LIN {X 0,Y 468.633,Z 235.957,A -85,B 0,C 180,E1 -7687.941,E2 -7687.941} C_VEL
LIN {X 0,Y 467.587,Z 230.243,A -85,B 0,C 180,E1 -7690.829,E2 -7690.829} C_VEL
LIN {X 0,Y 467.551,Z 230.247,A -85,B 0,C 180,E1 -7693.819,E2 -7693.819} C_VEL
LIN {X 0,Y 467.553,Z 230.248,A -85,B 0,C 180,E1 -7696.254,E2 -7696.254} C_VEL
LIN {X 0,Y 467.577,Z 230.245,A -85,B 0,C 180,E1 -7698.722,E2 -7698.722} C_VEL
LIN {X 0,Y 467.564,Z 230.246,A -85,B 0,C 180,E1 -7701.954,E2 -7701.954} C_VEL
LIN {X 0,Y 467.566,Z 230.245,A -85,B 0,C 180,E1 -7705.166,E2 -7705.166} C_VEL
LIN {X 0,Y 467.581,Z 230.243,A -85,B 0,C 180,E1 -7708.259,E2 -7708.259} C_VEL
LIN {X 0,Y 467.575,Z 230.245,A -85,B 0,C 180,E1 -7711.249,E2 -7711.249} C_VEL
LIN {X 0,Y 467.61,Z 230.239,A -85,B 0,C 180,E1 -7713.198,E2 -7713.198} C_VEL
LIN {X 0,Y 467.587,Z 230.242,A -85,B 0,C 180,E1 -7716.467,E2 -7716.467} C_VEL
LIN {X 0,Y 467.621,Z 230.237,A -85,B 0,C 180,E1 -7719.776,E2 -7719.776} C_VEL
LIN {X 0,Y 467.605,Z 230.241,A -85,B 0,C 180,E1 -7722.505,E2 -7722.505} C_VEL
LIN {X 0,Y 467.603,Z 230.24,A -85,B 0,C 180,E1 -7725.195,E2 -7725.195} C_VEL
LIN {X 0,Y 467.679,Z 230.23,A -85,B 0,C 180,E1 -7727.854,E2 -7727.854} C_VEL
LIN {X 0,Y 467.677,Z 230.231,A -85,B 0,C 180,E1 -7731.356,E2 -7731.356} C_VEL
LIN {X 0,Y 467.739,Z 230.225,A -85,B 0,C 180,E1 -7733.961,E2 -7733.961} C_VEL
LIN {X 0,Y 467.855,Z 230.21,A -85,B 0,C 180,E1 -7737.416,E2 -7737.416} C_VEL
LIN {X 0,Y 467.876,Z 230.206,A -85,B 0,C 180,E1 -7739.999,E2 -7739.999} C_VEL
LIN {X 0,Y 467.855,Z 230.208,A -85,B 0,C 180,E1 -7742.582,E2 -7742.582} C_VEL
LIN {X 0,Y 467.737,Z 230.224,A -85,B 0,C 180,E1 -7746.036,E2 -7746.036} C_VEL
LIN {X 0,Y 467.676,Z 230.232,A -85,B 0,C 180,E1 -7748.641,E2 -7748.641} C_VEL
LIN {X 0,Y 467.682,Z 230.231,A -85,B 0,C 180,E1 -7752.378,E2 -7752.378} C_VEL
LIN {X 0,Y 467.639,Z 230.239,A -85,B 0,C 180,E1 -7755.884,E2 -7755.884} C_VEL
LIN {X 0,Y 467.425,Z 230.265,A -85,B 0,C 180,E1 -7758.698,E2 -7758.698} C_VEL
LIN {X 0,Y 467.242,Z 230.477,A -85,B 0,C 180,E1 -7760.238,E2 -7760.238} C_VEL
LIN {X 0,Y 467.196,Z 233.681,A -85,B 0,C 180,E1 -7763.422,E2 -7763.422} C_VEL
LIN {X 0,Y 467.086,Z 236.163,A -85,B 0,C 180,E1 -7765.869,E2 -7765.869} C_VEL
LIN {X 0,Y 467.03,Z 239.651,A -85,B 0,C 180,E1 -7769.216,E2 -7769.216} C_VEL
LIN {X 0,Y 466.954,Z 242.322,A -85,B 0,C 180,E1 -7771.786,E2 -7771.786} C_VEL
LIN {X 0,Y 466.836,Z 245.609,A -85,B 0,C 180,E1 -7774.893,E2 -7774.893} C_VEL
LIN {X 0,Y 466.815,Z 248.588,A -85,B 0,C 180,E1 -7777.682,E2 -7777.682} C_VEL
LIN {X 0,Y 470.307,Z 263.21,A -85,B 0,C 180,E1 -7778.274,E2 -7778.274} C_VEL
LIN {X 0,Y 470.1,Z 275.079,A -85,B 0,C 180,E1 -7778.817,E2 -7778.817} C_VEL
LIN {X 0,Y 469.595,Z 287.366,A -85,B 0,C 180,E1 -7779.565,E2 -7779.565} C_VEL
LIN {X 0,Y 469.105,Z 298.069,A -85,B 0,C 180,E1 -7780.398,E2 -7780.398} C_VEL
LIN {X 0,Y 468.677,Z 308.639,A -85,B 0,C 180,E1 -7781.431,E2 -7781.431} C_VEL
LIN {X 0,Y 468.115,Z 318.546,A -85,B 0,C 180,E1 -7782.639,E2 -7782.639} C_VEL
LIN {X 0,Y 467.709,Z 326.533,A -85,B 0,C 180,E1 -7783.842,E2 -7783.842} C_VEL
LIN {X 0,Y 467.423,Z 332.988,A -85,B 0,C 180,E1 -7785.036,E2 -7785.036} C_VEL
LIN {X 0,Y 467.098,Z 339.332,A -85,B 0,C 180,E1 -7786.517,E2 -7786.517} C_VEL
LIN {X 0,Y 466.899,Z 344.209,A -85,B 0,C 180,E1 -7788.019,E2 -7788.019} C_VEL
LIN {X 0,Y 466.732,Z 347.944,A -85,B 0,C 180,E1 -7789.649,E2 -7789.649} C_VEL
LIN {X 0,Y 466.651,Z 349.597,A -85,B 0,C 180,E1 -7790.763,E2 -7790.763} C_VEL
LIN {X 0,Y 466.585,Z 350.586,A -85,B 0,C 180,E1 -7791.863,E2 -7791.863} C_VEL
LIN {X 0,Y 466.563,Z 350.949,A -85,B 0,C 180,E1 -7792.97,E2 -7792.97} C_VEL
LIN {X 0,Y 466.58,Z 350.427,A -85,B 0,C 180,E1 -7794.425,E2 -7794.425} C_VEL
LIN {X 0,Y 466.705,Z 348.328,A -85,B 0,C 180,E1 -7796.141,E2 -7796.141} C_VEL
LIN {X 0,Y 466.812,Z 345.614,A -85,B 0,C 180,E1 -7797.465,E2 -7797.465} C_VEL
LIN {X 0,Y 467.018,Z 340.95,A -85,B 0,C 180,E1 -7799.064,E2 -7799.064} C_VEL
LIN {X 0,Y 467.287,Z 335.172,A -85,B 0,C 180,E1 -7800.522,E2 -7800.522} C_VEL
LIN {X 0,Y 467.632,Z 327.673,A -85,B 0,C 180,E1 -7801.989,E2 -7801.989} C_VEL
LIN {X 0,Y 468.024,Z 319.77,A -85,B 0,C 180,E1 -7803.226,E2 -7803.226} C_VEL
LIN {X 0,Y 468.415,Z 311.541,A -85,B 0,C 180,E1 -7804.279,E2 -7804.279} C_VEL
LIN {X 0,Y 468.893,Z 301.772,A -85,B 0,C 180,E1 -7805.3,E2 -7805.3} C_VEL
LIN {X 0,Y 469.394,Z 290.021,A -85,B 0,C 180,E1 -7806.286,E2 -7806.286} C_VEL
LIN {X 0,Y 469.167,Z 284.982,A -85,B 0,C 180,E1 -7806.654,E2 -7806.654} C_VEL
LIN {X 0,Y 467.195,Z 276.584,A -85,B 0,C 180,E1 -7807.24,E2 -7807.24} C_VEL
LIN {X 0,Y 465.004,Z 269.763,A -85,B 0,C 180,E1 -7807.668,E2 -7807.668} C_VEL
LIN {X 0,Y 463.062,Z 262.658,A -85,B 0,C 180,E1 -7808.038,E2 -7808.038} C_VEL
LIN {X 0,Y 460.055,Z 249.852,A -85,B 0,C 180,E1 -7808.552,E2 -7808.552} C_VEL
LIN {X 0,Y 459.77,Z 248.251,A -85,B 0,C 180,E1 -7808.628,E2 -7808.628} C_VEL
LIN {X 0,Y 459.812,Z 245.224,A -85,B 0,C 180,E1 -7811.37,E2 -7811.37} C_VEL
LIN {X 0,Y 459.898,Z 242.015,A -85,B 0,C 180,E1 -7814.303,E2 -7814.303} C_VEL
LIN {X 0,Y 459.964,Z 238.118,A -85,B 0,C 180,E1 -7817.918,E2 -7817.918} C_VEL
LIN {X 0,Y 460.035,Z 234.635,A -85,B 0,C 180,E1 -7821.213,E2 -7821.213} C_VEL
LIN {X 0,Y 460.077,Z 231.831,A -85,B 0,C 180,E1 -7823.863,E2 -7823.863} C_VEL
LIN {X 0,Y 460.173,Z 231.168,A -85,B 0,C 180,E1 -7824.743,E2 -7824.743} C_VEL
LIN {X 0,Y 460.662,Z 231.104,A -85,B 0,C 180,E1 -7828.252,E2 -7828.252} C_VEL
LIN {X 0,Y 460.837,Z 231.082,A -85,B 0,C 180,E1 -7830.001,E2 -7830.001} C_VEL
LIN {X 0,Y 460.812,Z 231.084,A -85,B 0,C 180,E1 -7832.623,E2 -7832.623} C_VEL
LIN {X 0,Y 460.696,Z 231.099,A -85,B 0,C 180,E1 -7836.131,E2 -7836.131} C_VEL
LIN {X 0,Y 460.617,Z 231.111,A -85,B 0,C 180,E1 -7838.777,E2 -7838.777} C_VEL
LIN {X 0,Y 460.62,Z 231.109,A -85,B 0,C 180,E1 -7842.458,E2 -7842.458} C_VEL
LIN {X 0,Y 460.587,Z 231.111,A -85,B 0,C 180,E1 -7845.999,E2 -7845.999} C_VEL
LIN {X 0,Y 460.559,Z 231.119,A -85,B 0,C 180,E1 -7848.903,E2 -7848.903} C_VEL
LIN {X 0,Y 460.549,Z 231.118,A -85,B 0,C 180,E1 -7851.485,E2 -7851.485} C_VEL
LIN {X 0,Y 460.533,Z 231.119,A -85,B 0,C 180,E1 -7854.334,E2 -7854.334} C_VEL
LIN {X 0,Y 460.573,Z 231.115,A -85,B 0,C 180,E1 -7857.245,E2 -7857.245} C_VEL
LIN {X 0,Y 460.501,Z 231.124,A -85,B 0,C 180,E1 -7860.242,E2 -7860.242} C_VEL
LIN {X 0,Y 460.52,Z 231.122,A -85,B 0,C 180,E1 -7863.327,E2 -7863.327} C_VEL
LIN {X 0,Y 460.471,Z 231.129,A -85,B 0,C 180,E1 -7866.531,E2 -7866.531} C_VEL
LIN {X 0,Y 460.569,Z 231.115,A -85,B 0,C 180,E1 -7869.86,E2 -7869.86} C_VEL
LIN {X 0,Y 460.536,Z 231.121,A -85,B 0,C 180,E1 -7872.906,E2 -7872.906} C_VEL
LIN {X 0,Y 460.506,Z 231.123,A -85,B 0,C 180,E1 -7875.832,E2 -7875.832} C_VEL
LIN {X 0,Y 460.535,Z 231.12,A -85,B 0,C 180,E1 -7878.992,E2 -7878.992} C_VEL
LIN {X 0,Y 460.543,Z 231.117,A -85,B 0,C 180,E1 -7881.271,E2 -7881.271} C_VEL
LIN {X 0,Y 460.51,Z 231.124,A -85,B 0,C 180,E1 -7884.557,E2 -7884.557} C_VEL
LIN {X 0,Y 460.53,Z 231.12,A -85,B 0,C 180,E1 -7887.718,E2 -7887.718} C_VEL
LIN {X 0,Y 460.539,Z 231.12,A -85,B 0,C 180,E1 -7890.771,E2 -7890.771} C_VEL
LIN {X 0,Y 460.556,Z 231.118,A -85,B 0,C 180,E1 -7893.736,E2 -7893.736} C_VEL
LIN {X 0,Y 460.545,Z 231.12,A -85,B 0,C 180,E1 -7896.626,E2 -7896.626} C_VEL
LIN {X 0,Y 460.554,Z 231.118,A -85,B 0,C 180,E1 -7899.455,E2 -7899.455} C_VEL
LIN {X 0,Y 460.56,Z 231.118,A -85,B 0,C 180,E1 -7902.232,E2 -7902.232} C_VEL
LIN {X 0,Y 460.569,Z 231.115,A -85,B 0,C 180,E1 -7904.967,E2 -7904.967} C_VEL
LIN {X 0,Y 460.634,Z 231.109,A -85,B 0,C 180,E1 -7907.668,E2 -7907.668} C_VEL
LIN {X 0,Y 460.624,Z 231.108,A -85,B 0,C 180,E1 -7911.225,E2 -7911.225} C_VEL
LIN {X 0,Y 460.712,Z 231.099,A -85,B 0,C 180,E1 -7913.872,E2 -7913.872} C_VEL
LIN {X 0,Y 460.804,Z 231.086,A -85,B 0,C 180,E1 -7917.379,E2 -7917.379} C_VEL
LIN {X 0,Y 460.859,Z 231.081,A -85,B 0,C 180,E1 -7920.001,E2 -7920.001} C_VEL
LIN {X 0,Y 460.799,Z 231.085,A -85,B 0,C 180,E1 -7922.624,E2 -7922.624} C_VEL
LIN {X 0,Y 460.706,Z 231.099,A -85,B 0,C 180,E1 -7926.131,E2 -7926.131} C_VEL
LIN {X 0,Y 460.627,Z 231.107,A -85,B 0,C 180,E1 -7928.777,E2 -7928.777} C_VEL
LIN {X 0,Y 460.618,Z 231.109,A -85,B 0,C 180,E1 -7932.335,E2 -7932.335} C_VEL
LIN {X 0,Y 460.61,Z 231.11,A -85,B 0,C 180,E1 -7935.998,E2 -7935.998} C_VEL
LIN {X 0,Y 460.577,Z 231.116,A -85,B 0,C 180,E1 -7939.616,E2 -7939.616} C_VEL
LIN {X 0,Y 460.519,Z 231.12,A -85,B 0,C 180,E1 -7942.429,E2 -7942.429} C_VEL
LIN {X 0,Y 460.555,Z 231.118,A -85,B 0,C 180,E1 -7945.797,E2 -7945.797} C_VEL
LIN {X 0,Y 460.559,Z 231.116,A -85,B 0,C 180,E1 -7948.234,E2 -7948.234} C_VEL
LIN {X 0,Y 460.529,Z 231.121,A -85,B 0,C 180,E1 -7951.283,E2 -7951.283} C_VEL
LIN {X 0,Y 460.532,Z 231.121,A -85,B 0,C 180,E1 -7954.504,E2 -7954.504} C_VEL
LIN {X 0,Y 460.51,Z 231.123,A -85,B 0,C 180,E1 -7957.623,E2 -7957.623} C_VEL
LIN {X 0,Y 460.548,Z 231.119,A -85,B 0,C 180,E1 -7960.269,E2 -7960.269} C_VEL
LIN {X 0,Y 460.506,Z 231.125,A -85,B 0,C 180,E1 -7963.376,E2 -7963.376} C_VEL
LIN {X 0,Y 460.506,Z 231.122,A -85,B 0,C 180,E1 -7966.624,E2 -7966.624} C_VEL
LIN {X 0,Y 460.582,Z 231.165,A -85,B 0,C 180,E1 -7969.29,E2 -7969.29} C_VEL
LIN {X 0,Y 461.778,Z 238.038,A -85,B 0,C 180,E1 -7972.498,E2 -7972.498} C_VEL
LIN {X 0,Y 462.204,Z 241.909,A -85,B 0,C 180,E1 -7974.213,E2 -7974.213} C_VEL
LIN {X 0,Y 461.879,Z 248.185,A -85,B 0,C 180,E1 -7976.814,E2 -7976.814} C_VEL
LIN {X 0,Y 461.349,Z 256.833,A -85,B 0,C 180,E1 -7980.265,E2 -7980.265} C_VEL
LIN {X 0,Y 460.863,Z 265.93,A -85,B 0,C 180,E1 -7983.752,E2 -7983.752} C_VEL
LIN {X 0,Y 460.508,Z 274.929,A -85,B 0,C 180,E1 -7987.096,E2 -7987.096} C_VEL
LIN {X 0,Y 460.203,Z 283.998,A -85,B 0,C 180,E1 -7990.367,E2 -7990.367} C_VEL
LIN {X 0,Y 459.955,Z 294.33,A -85,B 0,C 180,E1 -7994.035,E2 -7994.035} C_VEL
LIN {X 0,Y 459.907,Z 295.245,A -85,B 0,C 180,E1 -7994.355,E2 -7994.355} C_VEL
LIN {X 0,Y 462.009,Z 310.185,A -85,B 0,C 180,E1 -7994.848,E2 -7994.848} C_VEL
LIN {X 0,Y 462.935,Z 318.538,A -85,B 0,C 180,E1 -7995.211,E2 -7995.211} C_VEL
LIN {X 0,Y 462.44,Z 330.386,A -85,B 0,C 180,E1 -7995.814,E2 -7995.814} C_VEL
LIN {X 0,Y 461.887,Z 341.871,A -85,B 0,C 180,E1 -7996.582,E2 -7996.582} C_VEL
LIN {X 0,Y 461.336,Z 353.209,A -85,B 0,C 180,E1 -7997.543,E2 -7997.543} C_VEL
LIN {X 0,Y 460.903,Z 362.933,A -85,B 0,C 180,E1 -7998.566,E2 -7998.566} C_VEL
LIN {X 0,Y 460.442,Z 371.517,A -85,B 0,C 180,E1 -7999.667,E2 -7999.667} C_VEL
LIN {X 0,Y 460.076,Z 379.873,A -85,B 0,C 180,E1 -8000.991,E2 -8000.991} C_VEL
LIN {X 0,Y 459.866,Z 386.614,A -85,B 0,C 180,E1 -8002.314,E2 -8002.314} C_VEL
LIN {X 0,Y 459.667,Z 392.79,A -85,B 0,C 180,E1 -8003.855,E2 -8003.855} C_VEL
LIN {X 0,Y 459.625,Z 396.799,A -85,B 0,C 180,E1 -8005.175,E2 -8005.175} C_VEL
LIN {X 0,Y 459.627,Z 399.756,A -85,B 0,C 180,E1 -8006.493,E2 -8006.493} C_VEL
LIN {X 0,Y 459.623,Z 401.165,A -85,B 0,C 180,E1 -8007.37,E2 -8007.37} C_VEL
LIN {X 0,Y 459.615,Z 402.164,A -85,B 0,C 180,E1 -8008.247,E2 -8008.247} C_VEL
LIN {X 0,Y 459.539,Z 402.977,A -85,B 0,C 180,E1 -8009.999,E2 -8009.999} C_VEL
LIN {X 0,Y 459.558,Z 402.751,A -85,B 0,C 180,E1 -8010.875,E2 -8010.875} C_VEL
LIN {X 0,Y 459.615,Z 402.128,A -85,B 0,C 180,E1 -8011.752,E2 -8011.752} C_VEL
LIN {X 0,Y 459.622,Z 401.11,A -85,B 0,C 180,E1 -8012.628,E2 -8012.628} C_VEL
LIN {X 0,Y 459.627,Z 399.686,A -85,B 0,C 180,E1 -8013.506,E2 -8013.506} C_VEL
LIN {X 0,Y 459.624,Z 396.696,A -85,B 0,C 180,E1 -8014.823,E2 -8014.823} C_VEL
LIN {X 0,Y 459.716,Z 391.613,A -85,B 0,C 180,E1 -8016.43,E2 -8016.43} C_VEL
LIN {X 0,Y 459.886,Z 385.437,A -85,B 0,C 180,E1 -8017.905,E2 -8017.905} C_VEL
LIN {X 0,Y 460.137,Z 378.45,A -85,B 0,C 180,E1 -8019.228,E2 -8019.228} C_VEL
LIN {X 0,Y 460.479,Z 369.718,A -85,B 0,C 180,E1 -8020.552,E2 -8020.552} C_VEL
LIN {X 0,Y 461,Z 360.789,A -85,B 0,C 180,E1 -8021.653,E2 -8021.653} C_VEL
LIN {X 0,Y 461.48,Z 349.763,A -85,B 0,C 180,E1 -8022.761,E2 -8022.761} C_VEL
LIN {X 0,Y 461.993,Z 338.756,A -85,B 0,C 180,E1 -8023.637,E2 -8023.637} C_VEL
LIN {X 0,Y 462.606,Z 326.426,A -85,B 0,C 180,E1 -8024.404,E2 -8024.404} C_VEL
LIN {X 0,Y 462.883,Z 317.395,A -85,B 0,C 180,E1 -8024.845,E2 -8024.845} C_VEL
LIN {X 0,Y 461.256,Z 303.73,A -85,B 0,C 180,E1 -8025.401,E2 -8025.401} C_VEL
LIN {X 0,Y 459.925,Z 294.533,A -85,B 0,C 180,E1 -8025.699,E2 -8025.699} C_VEL
LIN {X 0,Y 460.125,Z 284.742,A -85,B 0,C 180,E1 -8029.124,E2 -8029.124} C_VEL
LIN {X 0,Y 460.35,Z 276.829,A -85,B 0,C 180,E1 -8031.964,E2 -8031.964} C_VEL
LIN {X 0,Y 460.682,Z 267.815,A -85,B 0,C 180,E1 -8035.286,E2 -8035.286} C_VEL
LIN {X 0,Y 460.998,Z 260.214,A -85,B 0,C 180,E1 -8038.202,E2 -8038.202} C_VEL
LIN {X 0,Y 461.548,Z 251.983,A -85,B 0,C 180,E1 -8041.491,E2 -8041.491} C_VEL
LIN {X 0,Y 462.076,Z 244.167,A -85,B 0,C 180,E1 -8044.782,E2 -8044.782} C_VEL
LIN {X 0,Y 461.989,Z 239.448,A -85,B 0,C 180,E1 -8046.933,E2 -8046.933} C_VEL
LIN {X 0,Y 460.999,Z 233.637,A -85,B 0,C 180,E1 -8049.813,E2 -8049.813} C_VEL
LIN {X 0,Y 460.539,Z 231.121,A -85,B 0,C 180,E1 -8051.249,E2 -8051.249} C_VEL
LIN {X 0,Y 460.513,Z 231.125,A -85,B 0,C 180,E1 -8054.588,E2 -8054.588} C_VEL
LIN {X 0,Y 460.522,Z 231.124,A -85,B 0,C 180,E1 -8057.817,E2 -8057.817} C_VEL
LIN {X 0,Y 460.543,Z 231.121,A -85,B 0,C 180,E1 -8061.101,E2 -8061.101} C_VEL
LIN {X 0,Y 460.511,Z 231.126,A -85,B 0,C 180,E1 -8064.553,E2 -8064.553} C_VEL
LIN {X 0,Y 460.529,Z 231.123,A -85,B 0,C 180,E1 -8067.714,E2 -8067.714} C_VEL
LIN {X 0,Y 460.538,Z 231.12,A -85,B 0,C 180,E1 -8070.768,E2 -8070.768} C_VEL
LIN {X 0,Y 460.553,Z 231.119,A -85,B 0,C 180,E1 -8073.733,E2 -8073.733} C_VEL
LIN {X 0,Y 460.541,Z 231.12,A -85,B 0,C 180,E1 -8076.623,E2 -8076.623} C_VEL
LIN {X 0,Y 460.549,Z 231.119,A -85,B 0,C 180,E1 -8079.452,E2 -8079.452} C_VEL
LIN {X 0,Y 460.556,Z 231.118,A -85,B 0,C 180,E1 -8082.229,E2 -8082.229} C_VEL
LIN {X 0,Y 460.561,Z 231.119,A -85,B 0,C 180,E1 -8084.964,E2 -8084.964} C_VEL
LIN {X 0,Y 460.625,Z 231.109,A -85,B 0,C 180,E1 -8087.665,E2 -8087.665} C_VEL
LIN {X 0,Y 460.624,Z 231.109,A -85,B 0,C 180,E1 -8091.223,E2 -8091.223} C_VEL
LIN {X 0,Y 460.705,Z 231.101,A -85,B 0,C 180,E1 -8093.869,E2 -8093.869} C_VEL
LIN {X 0,Y 460.82,Z 231.087,A -85,B 0,C 180,E1 -8097.376,E2 -8097.376} C_VEL
LIN {X 0,Y 460.847,Z 231.082,A -85,B 0,C 180,E1 -8099.999,E2 -8099.999} C_VEL
LIN {X 0,Y 460.82,Z 231.085,A -85,B 0,C 180,E1 -8102.621,E2 -8102.621} C_VEL
LIN {X 0,Y 460.703,Z 231.1,A -85,B 0,C 180,E1 -8106.129,E2 -8106.129} C_VEL
LIN {X 0,Y 460.623,Z 231.11,A -85,B 0,C 180,E1 -8108.775,E2 -8108.775} C_VEL
LIN {X 0,Y 460.625,Z 231.11,A -85,B 0,C 180,E1 -8112.455,E2 -8112.455} C_VEL
LIN {X 0,Y 460.59,Z 231.117,A -85,B 0,C 180,E1 -8115.996,E2 -8115.996} C_VEL
LIN {X 0,Y 460.365,Z 231.144,A -85,B 0,C 180,E1 -8118.83,E2 -8118.83} C_VEL
LIN {X 0,Y 460.257,Z 231.158,A -85,B 0,C 180,E1 -8119.628,E2 -8119.628} C_VEL
LIN {X 0,Y 460.217,Z 232.417,A -85,B 0,C 180,E1 -8121.328,E2 -8121.328} C_VEL
LIN {X 0,Y 460.099,Z 235.425,A -85,B 0,C 180,E1 -8124.355,E2 -8124.355} C_VEL
LIN {X 0,Y 459.993,Z 238.744,A -85,B 0,C 180,E1 -8127.608,E2 -8127.608} C_VEL
LIN {X 0,Y 459.933,Z 241.517,A -85,B 0,C 180,E1 -8130.28,E2 -8130.28} C_VEL
LIN {X 0,Y 459.818,Z 244.726,A -85,B 0,C 180,E1 -8133.381,E2 -8133.381} C_VEL
LIN {X 0,Y 459.75,Z 248.134,A -85,B 0,C 180,E1 -8136.594,E2 -8136.594} C_VEL
LIN {X 0,Y 459.769,Z 249.036,A -85,B 0,C 180,E1 -8137.438,E2 -8137.438} C_VEL
LIN {X 0,Y 463.211,Z 263.105,A -85,B 0,C 180,E1 -8138.015,E2 -8138.015} C_VEL
LIN {X 0,Y 463.531,Z 266.233,A -85,B 0,C 180,E1 -8138.157,E2 -8138.157} C_VEL
LIN {X 0,Y 463.17,Z 278.071,A -85,B 0,C 180,E1 -8138.741,E2 -8138.741} C_VEL
LIN {X 0,Y 462.678,Z 288.478,A -85,B 0,C 180,E1 -8139.405,E2 -8139.405} C_VEL
LIN {X 0,Y 462.184,Z 299.123,A -85,B 0,C 180,E1 -8140.258,E2 -8140.258} C_VEL
LIN {X 0,Y 461.734,Z 309.41,A -85,B 0,C 180,E1 -8141.292,E2 -8141.292} C_VEL
LIN {X 0,Y 461.146,Z 319.156,A -85,B 0,C 180,E1 -8142.504,E2 -8142.504} C_VEL
LIN {X 0,Y 460.701,Z 327.31,A -85,B 0,C 180,E1 -8143.759,E2 -8143.759} C_VEL
LIN {X 0,Y 460.381,Z 333.775,A -85,B 0,C 180,E1 -8144.988,E2 -8144.988} C_VEL
LIN {X 0,Y 460.09,Z 339.048,A -85,B 0,C 180,E1 -8146.223,E2 -8146.223} C_VEL
LIN {X 0,Y 459.86,Z 344.077,A -85,B 0,C 180,E1 -8147.745,E2 -8147.745} C_VEL
LIN {X 0,Y 459.717,Z 346.989,A -85,B 0,C 180,E1 -8148.902,E2 -8148.902} C_VEL
LIN {X 0,Y 459.629,Z 349.08,A -85,B 0,C 180,E1 -8150.045,E2 -8150.045} C_VEL
LIN {X 0,Y 459.544,Z 350.542,A -85,B 0,C 180,E1 -8151.254,E2 -8151.254} C_VEL
LIN {X 0,Y 459.467,Z 351.304,A -85,B 0,C 180,E1 -8152.689,E2 -8152.689} C_VEL
LIN {X 0,Y 459.493,Z 350.807,A -85,B 0,C 180,E1 -8154.465,E2 -8154.465} C_VEL
LIN {X 0,Y 459.586,Z 349.516,A -85,B 0,C 180,E1 -8155.663,E2 -8155.663} C_VEL
LIN {X 0,Y 459.723,Z 346.737,A -85,B 0,C 180,E1 -8157.222,E2 -8157.222} C_VEL
LIN {X 0,Y 459.935,Z 342.363,A -85,B 0,C 180,E1 -8158.834,E2 -8158.834} C_VEL
LIN {X 0,Y 460.135,Z 337.57,A -85,B 0,C 180,E1 -8160.156,E2 -8160.156} C_VEL
LIN {X 0,Y 460.41,Z 331.357,A -85,B 0,C 180,E1 -8161.51,E2 -8161.51} C_VEL
LIN {X 0,Y 460.8,Z 324.163,A -85,B 0,C 180,E1 -8162.772,E2 -8162.772} C_VEL
LIN {X 0,Y 461.229,Z 315.329,A -85,B 0,C 180,E1 -8164.024,E2 -8164.024} C_VEL
LIN {X 0,Y 461.829,Z 305.53,A -85,B 0,C 180,E1 -8165.142,E2 -8165.142} C_VEL
LIN {X 0,Y 462.288,Z 294.927,A -85,B 0,C 180,E1 -8166.124,E2 -8166.124} C_VEL
LIN {X 0,Y 462.804,Z 283.147,A -85,B 0,C 180,E1 -8166.982,E2 -8166.982} C_VEL
LIN {X 0,Y 463.208,Z 271.238,A -85,B 0,C 180,E1 -8167.651,E2 -8167.651} C_VEL
LIN {X 0,Y 463.346,Z 263.971,A -85,B 0,C 180,E1 -8167.978,E2 -8167.978} C_VEL
LIN {X 0,Y 463.062,Z 262.658,A -85,B 0,C 180,E1 -8168.038,E2 -8168.038} C_VEL
LIN {X 0,Y 461.949,Z 260.691,A -85,B 0,C 180,E1 -8168.151,E2 -8168.151} C_VEL
LIN {X 0,Y 458.697,Z 258.451,A -85,B 0,C 180,E1 -8168.346,E2 -8168.346} C_VEL
LIN {X 0,Y 455.307,Z 256.242,A -85,B 0,C 180,E1 -8168.536,E2 -8168.536} C_VEL
LIN {X 0,Y 454.01,Z 254.292,A -85,B 0,C 180,E1 -8168.644,E2 -8168.644} C_VEL
LIN {X 0,Y 452.703,Z 248.622,A -85,B 0,C 180,E1 -8168.859,E2 -8168.859} C_VEL
LIN {X 0,Y 452.74,Z 245.271,A -85,B 0,C 180,E1 -8171.914,E2 -8171.914} C_VEL
LIN {X 0,Y 452.821,Z 242.262,A -85,B 0,C 180,E1 -8174.702,E2 -8174.702} C_VEL
LIN {X 0,Y 452.895,Z 238.339,A -85,B 0,C 180,E1 -8178.363,E2 -8178.363} C_VEL
LIN {X 0,Y 452.992,Z 234.514,A -85,B 0,C 180,E1 -8181.974,E2 -8181.974} C_VEL
LIN {X 0,Y 453.027,Z 232.657,A -85,B 0,C 180,E1 -8183.767,E2 -8183.767} C_VEL
LIN {X 0,Y 453.127,Z 232.045,A -85,B 0,C 180,E1 -8184.661,E2 -8184.661} C_VEL
LIN {X 0,Y 453.628,Z 231.98,A -85,B 0,C 180,E1 -8188.225,E2 -8188.225} C_VEL
LIN {X 0,Y 453.808,Z 231.957,A -85,B 0,C 180,E1 -8190.001,E2 -8190.001} C_VEL
LIN {X 0,Y 453.752,Z 231.963,A -85,B 0,C 180,E1 -8192.664,E2 -8192.664} C_VEL
LIN {X 0,Y 453.664,Z 231.975,A -85,B 0,C 180,E1 -8196.226,E2 -8196.226} C_VEL
LIN {X 0,Y 453.581,Z 231.988,A -85,B 0,C 180,E1 -8198.914,E2 -8198.914} C_VEL
LIN {X 0,Y 453.588,Z 231.985,A -85,B 0,C 180,E1 -8202.552,E2 -8202.552} C_VEL
LIN {X 0,Y 453.532,Z 231.99,A -85,B 0,C 180,E1 -8206.197,E2 -8206.197} C_VEL
LIN {X 0,Y 453.508,Z 231.997,A -85,B 0,C 180,E1 -8209.042,E2 -8209.042} C_VEL
LIN {X 0,Y 453.486,Z 231.997,A -85,B 0,C 180,E1 -8211.837,E2 -8211.837} C_VEL
LIN {X 0,Y 453.504,Z 231.998,A -85,B 0,C 180,E1 -8214.736,E2 -8214.736} C_VEL
LIN {X 0,Y 453.527,Z 231.992,A -85,B 0,C 180,E1 -8217.963,E2 -8217.963} C_VEL
LIN {X 0,Y 453.457,Z 232.001,A -85,B 0,C 180,E1 -8221.527,E2 -8221.527} C_VEL
LIN {X 0,Y 453.481,Z 232.001,A -85,B 0,C 180,E1 -8224.78,E2 -8224.78} C_VEL
LIN {X 0,Y 453.476,Z 232,A -85,B 0,C 180,E1 -8228.312,E2 -8228.312} C_VEL
LIN {X 0,Y 453.509,Z 231.997,A -85,B 0,C 180,E1 -8230.608,E2 -8230.608} C_VEL
LIN {X 0,Y 453.476,Z 231.998,A -85,B 0,C 180,E1 -8233.25,E2 -8233.25} C_VEL
LIN {X 0,Y 453.46,Z 232,A -85,B 0,C 180,E1 -8235.781,E2 -8235.781} C_VEL
LIN {X 0,Y 453.512,Z 231.993,A -85,B 0,C 180,E1 -8239.408,E2 -8239.408} C_VEL
LIN {X 0,Y 453.475,Z 232.002,A -85,B 0,C 180,E1 -8242.224,E2 -8242.224} C_VEL
LIN {X 0,Y 453.486,Z 231.997,A -85,B 0,C 180,E1 -8245.224,E2 -8245.224} C_VEL
LIN {X 0,Y 453.465,Z 232.002,A -85,B 0,C 180,E1 -8248.477,E2 -8248.477} C_VEL
LIN {X 0,Y 453.532,Z 231.993,A -85,B 0,C 180,E1 -8252.042,E2 -8252.042} C_VEL
LIN {X 0,Y 453.501,Z 231.994,A -85,B 0,C 180,E1 -8255.267,E2 -8255.267} C_VEL
LIN {X 0,Y 453.482,Z 231.999,A -85,B 0,C 180,E1 -8258.417,E2 -8258.417} C_VEL
LIN {X 0,Y 453.525,Z 231.991,A -85,B 0,C 180,E1 -8261.01,E2 -8261.01} C_VEL
LIN {X 0,Y 453.572,Z 231.989,A -85,B 0,C 180,E1 -8263.882,E2 -8263.882} C_VEL
LIN {X 0,Y 453.607,Z 231.984,A -85,B 0,C 180,E1 -8267.474,E2 -8267.474} C_VEL
LIN {X 0,Y 453.59,Z 231.984,A -85,B 0,C 180,E1 -8271.088,E2 -8271.088} C_VEL
LIN {X 0,Y 453.678,Z 231.975,A -85,B 0,C 180,E1 -8273.776,E2 -8273.776} C_VEL
LIN {X 0,Y 453.748,Z 231.965,A -85,B 0,C 180,E1 -8277.338,E2 -8277.338} C_VEL
LIN {X 0,Y 453.829,Z 231.956,A -85,B 0,C 180,E1 -8280.001,E2 -8280.001} C_VEL
LIN {X 0,Y 453.743,Z 231.964,A -85,B 0,C 180,E1 -8282.665,E2 -8282.665} C_VEL
LIN {X 0,Y 453.673,Z 231.975,A -85,B 0,C 180,E1 -8286.227,E2 -8286.227} C_VEL
LIN {X 0,Y 453.593,Z 231.984,A -85,B 0,C 180,E1 -8288.915,E2 -8288.915} C_VEL
LIN {X 0,Y 453.573,Z 231.986,A -85,B 0,C 180,E1 -8292.53,E2 -8292.53} C_VEL
LIN {X 0,Y 453.553,Z 231.988,A -85,B 0,C 180,E1 -8296.197,E2 -8296.197} C_VEL
LIN {X 0,Y 453.526,Z 231.993,A -85,B 0,C 180,E1 -8299.04,E2 -8299.04} C_VEL
LIN {X 0,Y 453.486,Z 231.998,A -85,B 0,C 180,E1 -8301.837,E2 -8301.837} C_VEL
LIN {X 0,Y 453.501,Z 231.995,A -85,B 0,C 180,E1 -8304.736,E2 -8304.736} C_VEL
LIN {X 0,Y 453.539,Z 231.991,A -85,B 0,C 180,E1 -8307.959,E2 -8307.959} C_VEL
LIN {X 0,Y 453.474,Z 232.001,A -85,B 0,C 180,E1 -8311.525,E2 -8311.525} C_VEL
LIN {X 0,Y 453.492,Z 231.998,A -85,B 0,C 180,E1 -8314.777,E2 -8314.777} C_VEL
LIN {X 0,Y 453.469,Z 231.999,A -85,B 0,C 180,E1 -8318.312,E2 -8318.312} C_VEL
LIN {X 0,Y 453.503,Z 231.996,A -85,B 0,C 180,E1 -8320.609,E2 -8320.609} C_VEL
LIN {X 0,Y 453.462,Z 232.003,A -85,B 0,C 180,E1 -8323.244,E2 -8323.244} C_VEL
LIN {X 0,Y 453.471,Z 231.999,A -85,B 0,C 180,E1 -8325.778,E2 -8325.778} C_VEL
LIN {X 0,Y 453.535,Z 232.068,A -85,B 0,C 180,E1 -8329.029,E2 -8329.029} C_VEL
LIN {X 0,Y 454.625,Z 238.376,A -85,B 0,C 180,E1 -8332.038,E2 -8332.038} C_VEL
LIN {X 0,Y 455.202,Z 242.871,A -85,B 0,C 180,E1 -8334.076,E2 -8334.076} C_VEL
LIN {X 0,Y 454.915,Z 248.685,A -85,B 0,C 180,E1 -8336.539,E2 -8336.539} C_VEL
LIN {X 0,Y 454.343,Z 257.275,A -85,B 0,C 180,E1 -8340.026,E2 -8340.026} C_VEL
LIN {X 0,Y 453.874,Z 265.669,A -85,B 0,C 180,E1 -8343.316,E2 -8343.316} C_VEL
LIN {X 0,Y 453.482,Z 274.636,A -85,B 0,C 180,E1 -8346.721,E2 -8346.721} C_VEL
LIN {X 0,Y 453.161,Z 283.64,A -85,B 0,C 180,E1 -8350.049,E2 -8350.049} C_VEL
LIN {X 0,Y 452.932,Z 292.682,A -85,B 0,C 180,E1 -8353.317,E2 -8353.317} C_VEL
LIN {X 0,Y 452.851,Z 294.962,A -85,B 0,C 180,E1 -8354.131,E2 -8354.131} C_VEL
LIN {X 0,Y 454.842,Z 308.85,A -85,B 0,C 180,E1 -8354.576,E2 -8354.576} C_VEL
LIN {X 0,Y 456,Z 319.27,A -85,B 0,C 180,E1 -8355.038,E2 -8355.038} C_VEL
LIN {X 0,Y 455.425,Z 331.663,A -85,B 0,C 180,E1 -8355.705,E2 -8355.705} C_VEL
LIN {X 0,Y 454.804,Z 344.24,A -85,B 0,C 180,E1 -8356.597,E2 -8356.597} C_VEL
LIN {X 0,Y 454.223,Z 355.309,A -85,B 0,C 180,E1 -8357.602,E2 -8357.602} C_VEL
LIN {X 0,Y 453.803,Z 364.308,A -85,B 0,C 180,E1 -8358.611,E2 -8358.611} C_VEL
LIN {X 0,Y 453.271,Z 374.07,A -85,B 0,C 180,E1 -8359.954,E2 -8359.954} C_VEL
LIN {X 0,Y 452.935,Z 381.873,A -85,B 0,C 180,E1 -8361.298,E2 -8361.298} C_VEL
LIN {X 0,Y 452.694,Z 389.043,A -85,B 0,C 180,E1 -8362.865,E2 -8362.865} C_VEL
LIN {X 0,Y 452.57,Z 393.818,A -85,B 0,C 180,E1 -8364.206,E2 -8364.206} C_VEL
LIN {X 0,Y 452.499,Z 397.466,A -85,B 0,C 180,E1 -8365.545,E2 -8365.545} C_VEL
LIN {X 0,Y 452.525,Z 399.351,A -85,B 0,C 180,E1 -8366.437,E2 -8366.437} C_VEL
LIN {X 0,Y 452.545,Z 400.763,A -85,B 0,C 180,E1 -8367.329,E2 -8367.329} C_VEL
LIN {X 0,Y 452.525,Z 401.763,A -85,B 0,C 180,E1 -8368.219,E2 -8368.219} C_VEL
LIN {X 0,Y 452.493,Z 402.368,A -85,B 0,C 180,E1 -8369.109,E2 -8369.109} C_VEL
LIN {X 0,Y 452.472,Z 402.579,A -85,B 0,C 180,E1 -8369.999,E2 -8369.999} C_VEL
LIN {X 0,Y 452.493,Z 402.355,A -85,B 0,C 180,E1 -8370.889,E2 -8370.889} C_VEL
LIN {X 0,Y 452.524,Z 401.731,A -85,B 0,C 180,E1 -8371.779,E2 -8371.779} C_VEL
LIN {X 0,Y 452.544,Z 400.712,A -85,B 0,C 180,E1 -8372.669,E2 -8372.669} C_VEL
LIN {X 0,Y 452.525,Z 399.287,A -85,B 0,C 180,E1 -8373.561,E2 -8373.561} C_VEL
LIN {X 0,Y 452.555,Z 396.299,A -85,B 0,C 180,E1 -8374.899,E2 -8374.899} C_VEL
LIN {X 0,Y 452.613,Z 391.718,A -85,B 0,C 180,E1 -8376.395,E2 -8376.395} C_VEL
LIN {X 0,Y 452.776,Z 386.066,A -85,B 0,C 180,E1 -8377.805,E2 -8377.805} C_VEL
LIN {X 0,Y 453.031,Z 379.304,A -85,B 0,C 180,E1 -8379.149,E2 -8379.149} C_VEL
LIN {X 0,Y 453.39,Z 370.931,A -85,B 0,C 180,E1 -8380.493,E2 -8380.493} C_VEL
LIN {X 0,Y 453.907,Z 362.371,A -85,B 0,C 180,E1 -8381.611,E2 -8381.611} C_VEL
LIN {X 0,Y 454.367,Z 352.234,A -85,B 0,C 180,E1 -8382.692,E2 -8382.692} C_VEL
LIN {X 0,Y 454.936,Z 341.394,A -85,B 0,C 180,E1 -8383.625,E2 -8383.625} C_VEL
LIN {X 0,Y 455.528,Z 330.018,A -85,B 0,C 180,E1 -8384.404,E2 -8384.404} C_VEL
LIN {X 0,Y 456.008,Z 318.41,A -85,B 0,C 180,E1 -8385.017,E2 -8385.017} C_VEL
LIN {X 0,Y 454.413,Z 304.619,A -85,B 0,C 180,E1 -8385.604,E2 -8385.604} C_VEL
LIN {X 0,Y 452.837,Z 294.155,A -85,B 0,C 180,E1 -8385.938,E2 -8385.938} C_VEL
LIN {X 0,Y 453.096,Z 284.254,A -85,B 0,C 180,E1 -8389.48,E2 -8389.48} C_VEL
LIN {X 0,Y 453.355,Z 275.233,A -85,B 0,C 180,E1 -8392.801,E2 -8392.801} C_VEL
LIN {X 0,Y 453.686,Z 266.654,A -85,B 0,C 180,E1 -8396.041,E2 -8396.041} C_VEL
LIN {X 0,Y 454.092,Z 258.699,A -85,B 0,C 180,E1 -8399.177,E2 -8399.177} C_VEL
LIN {X 0,Y 454.644,Z 251.344,A -85,B 0,C 180,E1 -8402.228,E2 -8402.228} C_VEL
LIN {X 0,Y 455.112,Z 244.802,A -85,B 0,C 180,E1 -8405.069,E2 -8405.069} C_VEL
LIN {X 0,Y 455.011,Z 240.563,A -85,B 0,C 180,E1 -8407.04,E2 -8407.04} C_VEL
LIN {X 0,Y 454.003,Z 234.765,A -85,B 0,C 180,E1 -8409.971,E2 -8409.971} C_VEL
LIN {X 0,Y 453.496,Z 231.997,A -85,B 0,C 180,E1 -8411.49,E2 -8411.49} C_VEL
LIN {X 0,Y 453.484,Z 232.001,A -85,B 0,C 180,E1 -8414.528,E2 -8414.528} C_VEL
LIN {X 0,Y 453.478,Z 232,A -85,B 0,C 180,E1 -8418.208,E2 -8418.208} C_VEL
LIN {X 0,Y 453.493,Z 231.999,A -85,B 0,C 180,E1 -8420.792,E2 -8420.792} C_VEL
LIN {X 0,Y 453.455,Z 232.003,A -85,B 0,C 180,E1 -8423.916,E2 -8423.916} C_VEL
LIN {X 0,Y 453.481,Z 231.999,A -85,B 0,C 180,E1 -8427.15,E2 -8427.15} C_VEL
LIN {X 0,Y 453.473,Z 232.002,A -85,B 0,C 180,E1 -8430.267,E2 -8430.267} C_VEL
LIN {X 0,Y 453.502,Z 231.997,A -85,B 0,C 180,E1 -8433.293,E2 -8433.293} C_VEL
LIN {X 0,Y 453.494,Z 231.997,A -85,B 0,C 180,E1 -8436.237,E2 -8436.237} C_VEL
LIN {X 0,Y 453.48,Z 232,A -85,B 0,C 180,E1 -8439.116,E2 -8439.116} C_VEL
LIN {X 0,Y 453.508,Z 231.995,A -85,B 0,C 180,E1 -8441.943,E2 -8441.943} C_VEL
LIN {X 0,Y 453.536,Z 231.992,A -85,B 0,C 180,E1 -8444.725,E2 -8444.725} C_VEL
LIN {X 0,Y 453.598,Z 231.985,A -85,B 0,C 180,E1 -8447.471,E2 -8447.471} C_VEL
LIN {X 0,Y 453.588,Z 231.986,A -85,B 0,C 180,E1 -8451.085,E2 -8451.085} C_VEL
LIN {X 0,Y 453.673,Z 231.976,A -85,B 0,C 180,E1 -8453.773,E2 -8453.773} C_VEL
LIN {X 0,Y 453.76,Z 231.966,A -85,B 0,C 180,E1 -8457.335,E2 -8457.335} C_VEL
LIN {X 0,Y 453.817,Z 231.957,A -85,B 0,C 180,E1 -8459.999,E2 -8459.999} C_VEL
LIN {X 0,Y 453.76,Z 231.964,A -85,B 0,C 180,E1 -8462.662,E2 -8462.662} C_VEL
LIN {X 0,Y 453.67,Z 231.977,A -85,B 0,C 180,E1 -8466.224,E2 -8466.224} C_VEL
LIN {X 0,Y 453.586,Z 231.986,A -85,B 0,C 180,E1 -8468.912,E2 -8468.912} C_VEL
LIN {X 0,Y 453.592,Z 231.986,A -85,B 0,C 180,E1 -8472.549,E2 -8472.549} C_VEL
LIN {X 0,Y 453.532,Z 231.996,A -85,B 0,C 180,E1 -8476.195,E2 -8476.195} C_VEL
LIN {X 0,Y 453.293,Z 232.025,A -85,B 0,C 180,E1 -8479,E2 -8479} C_VEL
LIN {X 0,Y 453.164,Z 232.042,A -85,B 0,C 180,E1 -8479.948,E2 -8479.948} C_VEL
LIN {X 0,Y 453.099,Z 234.75,A -85,B 0,C 180,E1 -8482.814,E2 -8482.814} C_VEL
LIN {X 0,Y 452.977,Z 237.744,A -85,B 0,C 180,E1 -8485.86,E2 -8485.86} C_VEL
LIN {X 0,Y 452.908,Z 240.71,A -85,B 0,C 180,E1 -8488.751,E2 -8488.751} C_VEL
LIN {X 0,Y 452.828,Z 243.876,A -85,B 0,C 180,E1 -8491.847,E2 -8491.847} C_VEL
LIN {X 0,Y 452.712,Z 247.218,A -85,B 0,C 180,E1 -8495.055,E2 -8495.055} C_VEL
LIN {X 0,Y 452.69,Z 249.429,A -85,B 0,C 180,E1 -8497.173,E2 -8497.173} C_VEL
LIN {X 0,Y 456.135,Z 263.437,A -85,B 0,C 180,E1 -8497.764,E2 -8497.764} C_VEL
LIN {X 0,Y 456.686,Z 267.165,A -85,B 0,C 180,E1 -8497.944,E2 -8497.944} C_VEL
LIN {X 0,Y 456.31,Z 278.804,A -85,B 0,C 180,E1 -8498.533,E2 -8498.533} C_VEL
LIN {X 0,Y 455.697,Z 290.811,A -85,B 0,C 180,E1 -8499.328,E2 -8499.328} C_VEL
LIN {X 0,Y 455.13,Z 302.258,A -85,B 0,C 180,E1 -8500.312,E2 -8500.312} C_VEL
LIN {X 0,Y 454.604,Z 312.682,A -85,B 0,C 180,E1 -8501.434,E2 -8501.434} C_VEL
LIN {X 0,Y 454.08,Z 320.978,A -85,B 0,C 180,E1 -8502.532,E2 -8502.532} C_VEL
LIN {X 0,Y 453.659,Z 328.716,A -85,B 0,C 180,E1 -8503.789,E2 -8503.789} C_VEL
LIN {X 0,Y 453.236,Z 336.231,A -85,B 0,C 180,E1 -8505.317,E2 -8505.317} C_VEL
LIN {X 0,Y 452.932,Z 341.961,A -85,B 0,C 180,E1 -8506.824,E2 -8506.824} C_VEL
LIN {X 0,Y 452.732,Z 345.851,A -85,B 0,C 180,E1 -8508.167,E2 -8508.167} C_VEL
LIN {X 0,Y 452.587,Z 348.761,A -85,B 0,C 180,E1 -8509.54,E2 -8509.54} C_VEL
LIN {X 0,Y 452.47,Z 350.708,A -85,B 0,C 180,E1 -8510.95,E2 -8510.95} C_VEL
LIN {X 0,Y 452.403,Z 351.707,A -85,B 0,C 180,E1 -8512.711,E2 -8512.711} C_VEL
LIN {X 0,Y 452.418,Z 351.548,A -85,B 0,C 180,E1 -8513.876,E2 -8513.876} C_VEL
LIN {X 0,Y 452.47,Z 350.285,A -85,B 0,C 180,E1 -8515.405,E2 -8515.405} C_VEL
LIN {X 0,Y 452.617,Z 347.536,A -85,B 0,C 180,E1 -8517.082,E2 -8517.082} C_VEL
LIN {X 0,Y 452.825,Z 343.732,A -85,B 0,C 180,E1 -8518.604,E2 -8518.604} C_VEL
LIN {X 0,Y 453.109,Z 337.827,A -85,B 0,C 180,E1 -8520.292,E2 -8520.292} C_VEL
LIN {X 0,Y 453.422,Z 331.446,A -85,B 0,C 180,E1 -8521.694,E2 -8521.694} C_VEL
LIN {X 0,Y 453.854,Z 323.585,A -85,B 0,C 180,E1 -8523.069,E2 -8523.069} C_VEL
LIN {X 0,Y 454.333,Z 314.532,A -85,B 0,C 180,E1 -8524.335,E2 -8524.335} C_VEL
LIN {X 0,Y 454.954,Z 304.651,A -85,B 0,C 180,E1 -8525.453,E2 -8525.453} C_VEL
LIN {X 0,Y 455.39,Z 294.999,A -85,B 0,C 180,E1 -8526.344,E2 -8526.344} C_VEL
LIN {X 0,Y 455.927,Z 283.116,A -85,B 0,C 180,E1 -8527.215,E2 -8527.215} C_VEL
LIN {X 0,Y 456.399,Z 270.783,A -85,B 0,C 180,E1 -8527.908,E2 -8527.908} C_VEL
LIN {X 0,Y 456.359,Z 264.561,A -85,B 0,C 180,E1 -8528.194,E2 -8528.194} C_VEL
LIN {X 0,Y 454.01,Z 254.292,A -85,B 0,C 180,E1 -8528.644,E2 -8528.644} C_VEL
LIN {X 0,Y 452.923,Z 251.776,A -85,B 0,C 180,E1 -8528.843,E2 -8528.843} C_VEL
LIN {X 0,Y 451.327,Z 249.568,A -85,B 0,C 180,E1 -8529.237,E2 -8529.237} C_VEL
LIN {X 0,Y 449.239,Z 247.919,A -85,B 0,C 180,E1 -8529.895,E2 -8529.895} C_VEL
LIN {X 0,Y 446.496,Z 246.612,A -85,B 0,C 180,E1 -8531.205,E2 -8531.205} C_VEL
LIN {X 0,Y 445.667,Z 245.502,A -85,B 0,C 180,E1 -8532.313,E2 -8532.313} C_VEL
LIN {X 0,Y 445.723,Z 242.192,A -85,B 0,C 180,E1 -8535.388,E2 -8535.388} C_VEL
LIN {X 0,Y 445.834,Z 239.231,A -85,B 0,C 180,E1 -8538.176,E2 -8538.176} C_VEL
LIN {X 0,Y 445.943,Z 235.376,A -85,B 0,C 180,E1 -8541.847,E2 -8541.847} C_VEL
LIN {X 0,Y 445.979,Z 233.496,A -85,B 0,C 180,E1 -8543.668,E2 -8543.668} C_VEL
LIN {X 0,Y 446.082,Z 232.922,A -85,B 0,C 180,E1 -8544.577,E2 -8544.577} C_VEL
LIN {X 0,Y 446.592,Z 232.856,A -85,B 0,C 180,E1 -8548.197,E2 -8548.197} C_VEL
LIN {X 0,Y 446.778,Z 232.833,A -85,B 0,C 180,E1 -8550.001,E2 -8550.001} C_VEL
LIN {X 0,Y 446.696,Z 232.842,A -85,B 0,C 180,E1 -8552.706,E2 -8552.706} C_VEL
LIN {X 0,Y 446.633,Z 232.851,A -85,B 0,C 180,E1 -8556.325,E2 -8556.325} C_VEL
LIN {X 0,Y 446.527,Z 232.866,A -85,B 0,C 180,E1 -8559.056,E2 -8559.056} C_VEL
LIN {X 0,Y 446.521,Z 232.866,A -85,B 0,C 180,E1 -8562.731,E2 -8562.731} C_VEL
LIN {X 0,Y 446.477,Z 232.87,A -85,B 0,C 180,E1 -8566.46,E2 -8566.46} C_VEL
LIN {X 0,Y 446.458,Z 232.874,A -85,B 0,C 180,E1 -8569.305,E2 -8569.305} C_VEL
LIN {X 0,Y 446.422,Z 232.877,A -85,B 0,C 180,E1 -8572.2,E2 -8572.2} C_VEL
LIN {X 0,Y 446.448,Z 232.875,A -85,B 0,C 180,E1 -8575.154,E2 -8575.154} C_VEL
LIN {X 0,Y 446.474,Z 232.871,A -85,B 0,C 180,E1 -8578.18,E2 -8578.18} C_VEL
LIN {X 0,Y 446.41,Z 232.878,A -85,B 0,C 180,E1 -8581.777,E2 -8581.777} C_VEL
LIN {X 0,Y 446.422,Z 232.879,A -85,B 0,C 180,E1 -8584.525,E2 -8584.525} C_VEL
LIN {X 0,Y 446.429,Z 232.876,A -85,B 0,C 180,E1 -8588.085,E2 -8588.085} C_VEL
LIN {X 0,Y 446.44,Z 232.876,A -85,B 0,C 180,E1 -8590.923,E2 -8590.923} C_VEL
LIN {X 0,Y 446.439,Z 232.874,A -85,B 0,C 180,E1 -8593.842,E2 -8593.842} C_VEL
LIN {X 0,Y 446.394,Z 232.883,A -85,B 0,C 180,E1 -8596.405,E2 -8596.405} C_VEL
LIN {X 0,Y 446.465,Z 232.872,A -85,B 0,C 180,E1 -8599.807,E2 -8599.807} C_VEL
LIN {X 0,Y 446.431,Z 232.878,A -85,B 0,C 180,E1 -8602.126,E2 -8602.126} C_VEL
LIN {X 0,Y 446.428,Z 232.876,A -85,B 0,C 180,E1 -8605.479,E2 -8605.479} C_VEL
LIN {X 0,Y 446.415,Z 232.88,A -85,B 0,C 180,E1 -8608.702,E2 -8608.702} C_VEL
LIN {X 0,Y 446.484,Z 232.87,A -85,B 0,C 180,E1 -8611.823,E2 -8611.823} C_VEL
LIN {X 0,Y 446.444,Z 232.874,A -85,B 0,C 180,E1 -8614.849,E2 -8614.849} C_VEL
LIN {X 0,Y 446.45,Z 232.876,A -85,B 0,C 180,E1 -8618.247,E2 -8618.247} C_VEL
LIN {X 0,Y 446.459,Z 232.874,A -85,B 0,C 180,E1 -8621.651,E2 -8621.651} C_VEL
LIN {X 0,Y 446.511,Z 232.867,A -85,B 0,C 180,E1 -8624.482,E2 -8624.482} C_VEL
LIN {X 0,Y 446.543,Z 232.865,A -85,B 0,C 180,E1 -8628.195,E2 -8628.195} C_VEL
LIN {X 0,Y 446.538,Z 232.862,A -85,B 0,C 180,E1 -8630.946,E2 -8630.946} C_VEL
LIN {X 0,Y 446.646,Z 232.851,A -85,B 0,C 180,E1 -8633.678,E2 -8633.678} C_VEL
LIN {X 0,Y 446.695,Z 232.843,A -85,B 0,C 180,E1 -8637.296,E2 -8637.296} C_VEL
LIN {X 0,Y 446.799,Z 232.832,A -85,B 0,C 180,E1 -8640.001,E2 -8640.001} C_VEL
LIN {X 0,Y 446.69,Z 232.842,A -85,B 0,C 180,E1 -8642.707,E2 -8642.707} C_VEL
LIN {X 0,Y 446.642,Z 232.85,A -85,B 0,C 180,E1 -8646.325,E2 -8646.325} C_VEL
LIN {X 0,Y 446.54,Z 232.863,A -85,B 0,C 180,E1 -8649.057,E2 -8649.057} C_VEL
LIN {X 0,Y 446.53,Z 232.864,A -85,B 0,C 180,E1 -8652.731,E2 -8652.731} C_VEL
LIN {X 0,Y 446.497,Z 232.866,A -85,B 0,C 180,E1 -8656.46,E2 -8656.46} C_VEL
LIN {X 0,Y 446.477,Z 232.873,A -85,B 0,C 180,E1 -8659.304,E2 -8659.304} C_VEL
LIN {X 0,Y 446.427,Z 232.876,A -85,B 0,C 180,E1 -8662.2,E2 -8662.2} C_VEL
LIN {X 0,Y 446.446,Z 232.877,A -85,B 0,C 180,E1 -8665.154,E2 -8665.154} C_VEL
LIN {X 0,Y 446.495,Z 232.868,A -85,B 0,C 180,E1 -8668.179,E2 -8668.179} C_VEL
LIN {X 0,Y 446.427,Z 232.877,A -85,B 0,C 180,E1 -8671.775,E2 -8671.775} C_VEL
LIN {X 0,Y 446.432,Z 232.877,A -85,B 0,C 180,E1 -8674.524,E2 -8674.524} C_VEL
LIN {X 0,Y 446.422,Z 232.876,A -85,B 0,C 180,E1 -8678.079,E2 -8678.079} C_VEL
LIN {X 0,Y 446.437,Z 232.876,A -85,B 0,C 180,E1 -8681.391,E2 -8681.391} C_VEL
LIN {X 0,Y 446.46,Z 232.871,A -85,B 0,C 180,E1 -8685.104,E2 -8685.104} C_VEL
LIN {X 0,Y 446.485,Z 232.945,A -85,B 0,C 180,E1 -8688.76,E2 -8688.76} C_VEL
LIN {X 0,Y 447.72,Z 240.152,A -85,B 0,C 180,E1 -8692.251,E2 -8692.251} C_VEL
LIN {X 0,Y 448.201,Z 243.915,A -85,B 0,C 180,E1 -8693.983,E2 -8693.983} C_VEL
LIN {X 0,Y 447.857,Z 250.199,A -85,B 0,C 180,E1 -8696.684,E2 -8696.684} C_VEL
LIN {X 0,Y 447.272,Z 259.043,A -85,B 0,C 180,E1 -8700.332,E2 -8700.332} C_VEL
LIN {X 0,Y 446.739,Z 267.934,A -85,B 0,C 180,E1 -8703.864,E2 -8703.864} C_VEL
LIN {X 0,Y 446.334,Z 276.881,A -85,B 0,C 180,E1 -8707.307,E2 -8707.307} C_VEL
LIN {X 0,Y 446.024,Z 285.874,A -85,B 0,C 180,E1 -8710.676,E2 -8710.676} C_VEL
LIN {X 0,Y 445.806,Z 294.589,A -85,B 0,C 180,E1 -8713.883,E2 -8713.883} C_VEL
LIN {X 0,Y 447.794,Z 308.426,A -85,B 0,C 180,E1 -8714.336,E2 -8714.336} C_VEL
LIN {X 0,Y 449.069,Z 319.867,A -85,B 0,C 180,E1 -8714.86,E2 -8714.86} C_VEL
LIN {X 0,Y 448.419,Z 332.89,A -85,B 0,C 180,E1 -8715.592,E2 -8715.592} C_VEL
LIN {X 0,Y 447.873,Z 343.735,A -85,B 0,C 180,E1 -8716.385,E2 -8716.385} C_VEL
LIN {X 0,Y 447.256,Z 354.835,A -85,B 0,C 180,E1 -8717.406,E2 -8717.406} C_VEL
LIN {X 0,Y 446.731,Z 365.644,A -85,B 0,C 180,E1 -8718.658,E2 -8718.658} C_VEL
LIN {X 0,Y 446.22,Z 373.624,A -85,B 0,C 180,E1 -8719.793,E2 -8719.793} C_VEL
LIN {X 0,Y 445.857,Z 381.442,A -85,B 0,C 180,E1 -8721.158,E2 -8721.158} C_VEL
LIN {X 0,Y 445.617,Z 388.619,A -85,B 0,C 180,E1 -8722.751,E2 -8722.751} C_VEL
LIN {X 0,Y 445.491,Z 392.834,A -85,B 0,C 180,E1 -8723.934,E2 -8723.934} C_VEL
LIN {X 0,Y 445.424,Z 397.056,A -85,B 0,C 180,E1 -8725.474,E2 -8725.474} C_VEL
LIN {X 0,Y 445.426,Z 398.942,A -85,B 0,C 180,E1 -8726.381,E2 -8726.381} C_VEL
LIN {X 0,Y 445.468,Z 400.36,A -85,B 0,C 180,E1 -8727.286,E2 -8727.286} C_VEL
LIN {X 0,Y 445.43,Z 401.968,A -85,B 0,C 180,E1 -8729.095,E2 -8729.095} C_VEL
LIN {X 0,Y 445.408,Z 402.181,A -85,B 0,C 180,E1 -8729.999,E2 -8729.999} C_VEL
LIN {X 0,Y 445.43,Z 401.959,A -85,B 0,C 180,E1 -8730.903,E2 -8730.903} C_VEL
LIN {X 0,Y 445.468,Z 400.316,A -85,B 0,C 180,E1 -8732.712,E2 -8732.712} C_VEL
LIN {X 0,Y 445.425,Z 398.89,A -85,B 0,C 180,E1 -8733.618,E2 -8733.618} C_VEL
LIN {X 0,Y 445.486,Z 395.904,A -85,B 0,C 180,E1 -8734.977,E2 -8734.977} C_VEL
LIN {X 0,Y 445.557,Z 390.417,A -85,B 0,C 180,E1 -8736.748,E2 -8736.748} C_VEL
LIN {X 0,Y 445.751,Z 384.65,A -85,B 0,C 180,E1 -8738.157,E2 -8738.157} C_VEL
LIN {X 0,Y 446.037,Z 377.668,A -85,B 0,C 180,E1 -8739.522,E2 -8739.522} C_VEL
LIN {X 0,Y 446.48,Z 368.953,A -85,B 0,C 180,E1 -8740.887,E2 -8740.887} C_VEL
LIN {X 0,Y 447.011,Z 360.036,A -85,B 0,C 180,E1 -8742.023,E2 -8742.023} C_VEL
LIN {X 0,Y 447.523,Z 349.938,A -85,B 0,C 180,E1 -8743.078,E2 -8743.078} C_VEL
LIN {X 0,Y 448.083,Z 339.629,A -85,B 0,C 180,E1 -8743.953,E2 -8743.953} C_VEL
LIN {X 0,Y 448.735,Z 327.813,A -85,B 0,C 180,E1 -8744.743,E2 -8744.743} C_VEL
LIN {X 0,Y 448.953,Z 318.184,A -85,B 0,C 180,E1 -8745.258,E2 -8745.258} C_VEL
LIN {X 0,Y 447.417,Z 304.538,A -85,B 0,C 180,E1 -8745.855,E2 -8745.855} C_VEL
LIN {X 0,Y 445.791,Z 293.706,A -85,B 0,C 180,E1 -8746.23,E2 -8746.23} C_VEL
LIN {X 0,Y 446.05,Z 283.921,A -85,B 0,C 180,E1 -8749.8,E2 -8749.8} C_VEL
LIN {X 0,Y 446.328,Z 274.94,A -85,B 0,C 180,E1 -8753.181,E2 -8753.181} C_VEL
LIN {X 0,Y 446.677,Z 267.027,A -85,B 0,C 180,E1 -8756.253,E2 -8756.253} C_VEL
LIN {X 0,Y 447.165,Z 258.547,A -85,B 0,C 180,E1 -8759.674,E2 -8759.674} C_VEL
LIN {X 0,Y 447.727,Z 251.205,A -85,B 0,C 180,E1 -8762.788,E2 -8762.788} C_VEL
LIN {X 0,Y 448.141,Z 245.191,A -85,B 0,C 180,E1 -8765.467,E2 -8765.467} C_VEL
LIN {X 0,Y 448.069,Z 242.234,A -85,B 0,C 180,E1 -8766.874,E2 -8766.874} C_VEL
LIN {X 0,Y 447.15,Z 236.851,A -85,B 0,C 180,E1 -8769.632,E2 -8769.632} C_VEL
LIN {X 0,Y 446.444,Z 232.876,A -85,B 0,C 180,E1 -8771.84,E2 -8771.84} C_VEL
LIN {X 0,Y 446.451,Z 232.876,A -85,B 0,C 180,E1 -8775.102,E2 -8775.102} C_VEL
LIN {X 0,Y 446.427,Z 232.879,A -85,B 0,C 180,E1 -8778.608,E2 -8778.608} C_VEL
LIN {X 0,Y 446.444,Z 232.878,A -85,B 0,C 180,E1 -8780.972,E2 -8780.972} C_VEL
LIN {X 0,Y 446.419,Z 232.881,A -85,B 0,C 180,E1 -8784.373,E2 -8784.373} C_VEL
LIN {X 0,Y 446.42,Z 232.88,A -85,B 0,C 180,E1 -8787.637,E2 -8787.637} C_VEL
LIN {X 0,Y 446.447,Z 232.875,A -85,B 0,C 180,E1 -8790.789,E2 -8790.789} C_VEL
LIN {X 0,Y 446.475,Z 232.872,A -85,B 0,C 180,E1 -8793.847,E2 -8793.847} C_VEL
LIN {X 0,Y 446.423,Z 232.88,A -85,B 0,C 180,E1 -8796.822,E2 -8796.822} C_VEL
LIN {X 0,Y 446.441,Z 232.875,A -85,B 0,C 180,E1 -8799.736,E2 -8799.736} C_VEL
LIN {X 0,Y 446.46,Z 232.875,A -85,B 0,C 180,E1 -8802.596,E2 -8802.596} C_VEL
LIN {X 0,Y 446.466,Z 232.872,A -85,B 0,C 180,E1 -8805.411,E2 -8805.411} C_VEL
LIN {X 0,Y 446.535,Z 232.866,A -85,B 0,C 180,E1 -8808.192,E2 -8808.192} C_VEL
LIN {X 0,Y 446.595,Z 232.858,A -85,B 0,C 180,E1 -8811.856,E2 -8811.856} C_VEL
LIN {X 0,Y 446.641,Z 232.85,A -85,B 0,C 180,E1 -8814.581,E2 -8814.581} C_VEL
LIN {X 0,Y 446.704,Z 232.844,A -85,B 0,C 180,E1 -8817.293,E2 -8817.293} C_VEL
LIN {X 0,Y 446.788,Z 232.833,A -85,B 0,C 180,E1 -8819.999,E2 -8819.999} C_VEL
LIN {X 0,Y 446.704,Z 232.844,A -85,B 0,C 180,E1 -8822.704,E2 -8822.704} C_VEL
LIN {X 0,Y 446.64,Z 232.853,A -85,B 0,C 180,E1 -8826.322,E2 -8826.322} C_VEL
LIN {X 0,Y 446.532,Z 232.865,A -85,B 0,C 180,E1 -8829.054,E2 -8829.054} C_VEL
LIN {X 0,Y 446.526,Z 232.866,A -85,B 0,C 180,E1 -8832.728,E2 -8832.728} C_VEL
LIN {X 0,Y 446.503,Z 232.872,A -85,B 0,C 180,E1 -8836.234,E2 -8836.234} C_VEL
LIN {X 0,Y 446.2,Z 232.909,A -85,B 0,C 180,E1 -8839.314,E2 -8839.314} C_VEL
LIN {X 0,Y 446.096,Z 233.141,A -85,B 0,C 180,E1 -8840.278,E2 -8840.278} C_VEL
LIN {X 0,Y 446.027,Z 235.962,A -85,B 0,C 180,E1 -8843.197,E2 -8843.197} C_VEL
LIN {X 0,Y 445.932,Z 238.891,A -85,B 0,C 180,E1 -8846.184,E2 -8846.184} C_VEL
LIN {X 0,Y 445.828,Z 242.009,A -85,B 0,C 180,E1 -8849.252,E2 -8849.252} C_VEL
LIN {X 0,Y 445.751,Z 245.185,A -85,B 0,C 180,E1 -8852.414,E2 -8852.414} C_VEL
LIN {X 0,Y 445.618,Z 248.604,A -85,B 0,C 180,E1 -8855.698,E2 -8855.698} C_VEL
LIN {X 0,Y 445.647,Z 249.848,A -85,B 0,C 180,E1 -8856.904,E2 -8856.904} C_VEL
LIN {X 0,Y 448.98,Z 263.29,A -85,B 0,C 180,E1 -8857.48,E2 -8857.48} C_VEL
LIN {X 0,Y 449.875,Z 268.062,A -85,B 0,C 180,E1 -8857.721,E2 -8857.721} C_VEL
LIN {X 0,Y 449.413,Z 280.405,A -85,B 0,C 180,E1 -8858.366,E2 -8858.366} C_VEL
LIN {X 0,Y 448.869,Z 290.679,A -85,B 0,C 180,E1 -8859.062,E2 -8859.062} C_VEL
LIN {X 0,Y 448.306,Z 301.549,A -85,B 0,C 180,E1 -8859.995,E2 -8859.995} C_VEL
LIN {X 0,Y 447.75,Z 311.99,A -85,B 0,C 180,E1 -8861.114,E2 -8861.114} C_VEL
LIN {X 0,Y 447.123,Z 321.494,A -85,B 0,C 180,E1 -8862.376,E2 -8862.376} C_VEL
LIN {X 0,Y 446.6,Z 330.101,A -85,B 0,C 180,E1 -8863.819,E2 -8863.819} C_VEL
LIN {X 0,Y 446.232,Z 336.381,A -85,B 0,C 180,E1 -8865.129,E2 -8865.129} C_VEL
LIN {X 0,Y 445.937,Z 341.505,A -85,B 0,C 180,E1 -8866.463,E2 -8866.463} C_VEL
LIN {X 0,Y 445.691,Z 345.591,A -85,B 0,C 180,E1 -8867.825,E2 -8867.825} C_VEL
LIN {X 0,Y 445.532,Z 348.676,A -85,B 0,C 180,E1 -8869.212,E2 -8869.212} C_VEL
LIN {X 0,Y 445.394,Z 351.068,A -85,B 0,C 180,E1 -8870.865,E2 -8870.865} C_VEL
LIN {X 0,Y 445.328,Z 351.943,A -85,B 0,C 180,E1 -8872.096,E2 -8872.096} C_VEL
LIN {X 0,Y 445.314,Z 352.046,A -85,B 0,C 180,E1 -8873.596,E2 -8873.596} C_VEL
LIN {X 0,Y 445.395,Z 350.74,A -85,B 0,C 180,E1 -8875.387,E2 -8875.387} C_VEL
LIN {X 0,Y 445.49,Z 348.738,A -85,B 0,C 180,E1 -8876.729,E2 -8876.729} C_VEL
LIN {X 0,Y 445.714,Z 344.988,A -85,B 0,C 180,E1 -8878.368,E2 -8878.368} C_VEL
LIN {X 0,Y 445.967,Z 339.483,A -85,B 0,C 180,E1 -8880.079,E2 -8880.079} C_VEL
LIN {X 0,Y 446.306,Z 333.146,A -85,B 0,C 180,E1 -8881.554,E2 -8881.554} C_VEL
LIN {X 0,Y 446.735,Z 326.146,A -85,B 0,C 180,E1 -8882.857,E2 -8882.857} C_VEL
LIN {X 0,Y 447.218,Z 317.631,A -85,B 0,C 180,E1 -8884.146,E2 -8884.146} C_VEL
LIN {X 0,Y 447.812,Z 308.608,A -85,B 0,C 180,E1 -8885.256,E2 -8885.256} C_VEL
LIN {X 0,Y 448.348,Z 297.929,A -85,B 0,C 180,E1 -8886.318,E2 -8886.318} C_VEL
LIN {X 0,Y 448.949,Z 286.221,A -85,B 0,C 180,E1 -8887.243,E2 -8887.243} C_VEL
LIN {X 0,Y 449.366,Z 274.65,A -85,B 0,C 180,E1 -8887.955,E2 -8887.955} C_VEL
LIN {X 0,Y 449.61,Z 266.292,A -85,B 0,C 180,E1 -8888.356,E2 -8888.356} C_VEL
LIN {X 0,Y 446.811,Z 254.004,A -85,B 0,C 180,E1 -8888.913,E2 -8888.913} C_VEL
LIN {X 0,Y 445.624,Z 248.991,A -85,B 0,C 180,E1 -8889.096,E2 -8889.096} C_VEL
LIN {X 0,Y 445.667,Z 245.502,A -85,B 0,C 180,E1 -8892.313,E2 -8892.313} C_VEL
LIN {X 0,Y 445.028,Z 244.765,A -85,B 0,C 180,E1 -8893.061,E2 -8893.061} C_VEL
LIN {X 0,Y 442.205,Z 243.723,A -85,B 0,C 180,E1 -8894.28,E2 -8894.28} C_VEL
LIN {X 0,Y 439.8,Z 242.9,A -85,B 0,C 180,E1 -8895.264,E2 -8895.264} C_VEL
LIN {X 0,Y 438.76,Z 242.195,A -85,B 0,C 180,E1 -8896.022,E2 -8896.022} C_VEL
LIN {X 0,Y 438.672,Z 241.932,A -85,B 0,C 180,E1 -8896.279,E2 -8896.279} C_VEL
LIN {X 0,Y 438.766,Z 239.158,A -85,B 0,C 180,E1 -8898.919,E2 -8898.919} C_VEL
LIN {X 0,Y 438.882,Z 236.255,A -85,B 0,C 180,E1 -8901.715,E2 -8901.715} C_VEL
LIN {X 0,Y 438.932,Z 234.361,A -85,B 0,C 180,E1 -8903.566,E2 -8903.566} C_VEL
LIN {X 0,Y 439.039,Z 233.799,A -85,B 0,C 180,E1 -8904.489,E2 -8904.489} C_VEL
LIN {X 0,Y 439.556,Z 233.732,A -85,B 0,C 180,E1 -8908.168,E2 -8908.168} C_VEL
LIN {X 0,Y 439.748,Z 233.709,A -85,B 0,C 180,E1 -8910.001,E2 -8910.001} C_VEL
LIN {X 0,Y 439.643,Z 233.721,A -85,B 0,C 180,E1 -8912.75,E2 -8912.75} C_VEL
LIN {X 0,Y 439.604,Z 233.726,A -85,B 0,C 180,E1 -8916.426,E2 -8916.426} C_VEL
LIN {X 0,Y 439.489,Z 233.742,A -85,B 0,C 180,E1 -8919.203,E2 -8919.203} C_VEL
LIN {X 0,Y 439.491,Z 233.741,A -85,B 0,C 180,E1 -8922.728,E2 -8922.728} C_VEL
LIN {X 0,Y 439.434,Z 233.746,A -85,B 0,C 180,E1 -8926.35,E2 -8926.35} C_VEL
LIN {X 0,Y 439.422,Z 233.75,A -85,B 0,C 180,E1 -8929.626,E2 -8929.626} C_VEL
LIN {X 0,Y 439.363,Z 233.758,A -85,B 0,C 180,E1 -8932.576,E2 -8932.576} C_VEL
LIN {X 0,Y 439.395,Z 233.753,A -85,B 0,C 180,E1 -8935.586,E2 -8935.586} C_VEL
LIN {X 0,Y 439.407,Z 233.753,A -85,B 0,C 180,E1 -8938.675,E2 -8938.675} C_VEL
LIN {X 0,Y 439.361,Z 233.756,A -85,B 0,C 180,E1 -8942.032,E2 -8942.032} C_VEL
LIN {X 0,Y 439.388,Z 233.753,A -85,B 0,C 180,E1 -8945.343,E2 -8945.343} C_VEL
LIN {X 0,Y 439.39,Z 233.756,A -85,B 0,C 180,E1 -8948.595,E2 -8948.595} C_VEL
LIN {X 0,Y 439.398,Z 233.753,A -85,B 0,C 180,E1 -8951.261,E2 -8951.261} C_VEL
LIN {X 0,Y 439.403,Z 233.753,A -85,B 0,C 180,E1 -8954.73,E2 -8954.73} C_VEL
LIN {X 0,Y 439.392,Z 233.753,A -85,B 0,C 180,E1 -8957.798,E2 -8957.798} C_VEL
LIN {X 0,Y 439.448,Z 233.748,A -85,B 0,C 180,E1 -8960.232,E2 -8960.232} C_VEL
LIN {X 0,Y 439.374,Z 233.755,A -85,B 0,C 180,E1 -8963.715,E2 -8963.715} C_VEL
LIN {X 0,Y 439.37,Z 233.755,A -85,B 0,C 180,E1 -8967.056,E2 -8967.056} C_VEL
LIN {X 0,Y 439.382,Z 233.757,A -85,B 0,C 180,E1 -8970.276,E2 -8970.276} C_VEL
LIN {X 0,Y 439.428,Z 233.748,A -85,B 0,C 180,E1 -8973.398,E2 -8973.398} C_VEL
LIN {X 0,Y 439.385,Z 233.755,A -85,B 0,C 180,E1 -8976.431,E2 -8976.431} C_VEL
LIN {X 0,Y 439.391,Z 233.753,A -85,B 0,C 180,E1 -8979.399,E2 -8979.399} C_VEL
LIN {X 0,Y 439.433,Z 233.75,A -85,B 0,C 180,E1 -8982.311,E2 -8982.311} C_VEL
LIN {X 0,Y 439.451,Z 233.745,A -85,B 0,C 180,E1 -8985.176,E2 -8985.176} C_VEL
LIN {X 0,Y 439.512,Z 233.74,A -85,B 0,C 180,E1 -8988.004,E2 -8988.004} C_VEL
LIN {X 0,Y 439.509,Z 233.74,A -85,B 0,C 180,E1 -8991.727,E2 -8991.727} C_VEL
LIN {X 0,Y 439.625,Z 233.723,A -85,B 0,C 180,E1 -8994.497,E2 -8994.497} C_VEL
LIN {X 0,Y 439.64,Z 233.723,A -85,B 0,C 180,E1 -8998.169,E2 -8998.169} C_VEL
LIN {X 0,Y 439.769,Z 233.708,A -85,B 0,C 180,E1 -9000.001,E2 -9000.001} C_VEL
LIN {X 0,Y 439.639,Z 233.72,A -85,B 0,C 180,E1 -9002.75,E2 -9002.75} C_VEL
LIN {X 0,Y 439.612,Z 233.725,A -85,B 0,C 180,E1 -9006.427,E2 -9006.427} C_VEL
LIN {X 0,Y 439.503,Z 233.741,A -85,B 0,C 180,E1 -9009.203,E2 -9009.203} C_VEL
LIN {X 0,Y 439.474,Z 233.743,A -85,B 0,C 180,E1 -9012.939,E2 -9012.939} C_VEL
LIN {X 0,Y 439.455,Z 233.743,A -85,B 0,C 180,E1 -9016.349,E2 -9016.349} C_VEL
LIN {X 0,Y 439.411,Z 233.752,A -85,B 0,C 180,E1 -9019.627,E2 -9019.627} C_VEL
LIN {X 0,Y 439.372,Z 233.754,A -85,B 0,C 180,E1 -9022.576,E2 -9022.576} C_VEL
LIN {X 0,Y 439.395,Z 233.754,A -85,B 0,C 180,E1 -9025.587,E2 -9025.587} C_VEL
LIN {X 0,Y 439.427,Z 233.749,A -85,B 0,C 180,E1 -9028.674,E2 -9028.674} C_VEL
LIN {X 0,Y 439.378,Z 233.754,A -85,B 0,C 180,E1 -9032.03,E2 -9032.03} C_VEL
LIN {X 0,Y 439.401,Z 233.754,A -85,B 0,C 180,E1 -9035.34,E2 -9035.34} C_VEL
LIN {X 0,Y 439.379,Z 233.755,A -85,B 0,C 180,E1 -9038.597,E2 -9038.597} C_VEL
LIN {X 0,Y 439.398,Z 233.754,A -85,B 0,C 180,E1 -9041.257,E2 -9041.257} C_VEL
LIN {X 0,Y 439.408,Z 233.75,A -85,B 0,C 180,E1 -9044.73,E2 -9044.73} C_VEL
LIN {X 0,Y 439.425,Z 233.855,A -85,B 0,C 180,E1 -9048.496,E2 -9048.496} C_VEL
LIN {X 0,Y 440.484,Z 239.934,A -85,B 0,C 180,E1 -9051.518,E2 -9051.518} C_VEL
LIN {X 0,Y 441.202,Z 244.961,A -85,B 0,C 180,E1 -9053.886,E2 -9053.886} C_VEL
LIN {X 0,Y 440.958,Z 249.96,A -85,B 0,C 180,E1 -9056.093,E2 -9056.093} C_VEL
LIN {X 0,Y 440.356,Z 257.522,A -85,B 0,C 180,E1 -9059.288,E2 -9059.288} C_VEL
LIN {X 0,Y 439.879,Z 265.108,A -85,B 0,C 180,E1 -9062.396,E2 -9062.396} C_VEL
LIN {X 0,Y 439.446,Z 273.506,A -85,B 0,C 180,E1 -9065.728,E2 -9065.728} C_VEL
LIN {X 0,Y 439.098,Z 281.678,A -85,B 0,C 180,E1 -9068.891,E2 -9068.891} C_VEL
LIN {X 0,Y 438.84,Z 289.345,A -85,B 0,C 180,E1 -9071.802,E2 -9071.802} C_VEL
LIN {X 0,Y 438.74,Z 294.212,A -85,B 0,C 180,E1 -9073.619,E2 -9073.619} C_VEL
LIN {X 0,Y 440.859,Z 308.877,A -85,B 0,C 180,E1 -9074.127,E2 -9074.127} C_VEL
LIN {X 0,Y 442.104,Z 321.525,A -85,B 0,C 180,E1 -9074.734,E2 -9074.734} C_VEL
LIN {X 0,Y 441.437,Z 334.101,A -85,B 0,C 180,E1 -9075.477,E2 -9075.477} C_VEL
LIN {X 0,Y 440.811,Z 345.372,A -85,B 0,C 180,E1 -9076.35,E2 -9076.35} C_VEL
LIN {X 0,Y 440.146,Z 356.493,A -85,B 0,C 180,E1 -9077.434,E2 -9077.434} C_VEL
LIN {X 0,Y 439.7,Z 365.168,A -85,B 0,C 180,E1 -9078.474,E2 -9078.474} C_VEL
LIN {X 0,Y 439.198,Z 373.164,A -85,B 0,C 180,E1 -9079.628,E2 -9079.628} C_VEL
LIN {X 0,Y 438.803,Z 380.999,A -85,B 0,C 180,E1 -9081.015,E2 -9081.015} C_VEL
LIN {X 0,Y 438.54,Z 388.187,A -85,B 0,C 180,E1 -9082.633,E2 -9082.633} C_VEL
LIN {X 0,Y 438.392,Z 392.84,A -85,B 0,C 180,E1 -9083.973,E2 -9083.973} C_VEL
LIN {X 0,Y 438.353,Z 396.642,A -85,B 0,C 180,E1 -9085.401,E2 -9085.401} C_VEL
LIN {X 0,Y 438.328,Z 398.531,A -85,B 0,C 180,E1 -9086.322,E2 -9086.322} C_VEL
LIN {X 0,Y 438.393,Z 399.955,A -85,B 0,C 180,E1 -9087.242,E2 -9087.242} C_VEL
LIN {X 0,Y 438.369,Z 401.568,A -85,B 0,C 180,E1 -9089.08,E2 -9089.08} C_VEL
LIN {X 0,Y 438.345,Z 401.783,A -85,B 0,C 180,E1 -9089.999,E2 -9089.999} C_VEL
LIN {X 0,Y 438.353,Z 401.564,A -85,B 0,C 180,E1 -9090.918,E2 -9090.918} C_VEL
LIN {X 0,Y 438.393,Z 399.923,A -85,B 0,C 180,E1 -9092.756,E2 -9092.756} C_VEL
LIN {X 0,Y 438.326,Z 398.497,A -85,B 0,C 180,E1 -9093.676,E2 -9093.676} C_VEL
LIN {X 0,Y 438.416,Z 395.514,A -85,B 0,C 180,E1 -9095.057,E2 -9095.057} C_VEL
LIN {X 0,Y 438.451,Z 391.478,A -85,B 0,C 180,E1 -9096.441,E2 -9096.441} C_VEL
LIN {X 0,Y 438.66,Z 385.292,A -85,B 0,C 180,E1 -9098.058,E2 -9098.058} C_VEL
LIN {X 0,Y 438.933,Z 378.541,A -85,B 0,C 180,E1 -9099.445,E2 -9099.445} C_VEL
LIN {X 0,Y 439.348,Z 370.186,A -85,B 0,C 180,E1 -9100.833,E2 -9100.833} C_VEL
LIN {X 0,Y 439.942,Z 361.654,A -85,B 0,C 180,E1 -9101.985,E2 -9101.985} C_VEL
LIN {X 0,Y 440.481,Z 351.426,A -85,B 0,C 180,E1 -9103.112,E2 -9103.112} C_VEL
LIN {X 0,Y 441.084,Z 340.761,A -85,B 0,C 180,E1 -9104.062,E2 -9104.062} C_VEL
LIN {X 0,Y 441.778,Z 329.455,A -85,B 0,C 180,E1 -9104.863,E2 -9104.863} C_VEL
LIN {X 0,Y 442.08,Z 319.142,A -85,B 0,C 180,E1 -9105.442,E2 -9105.442} C_VEL
LIN {X 0,Y 440.721,Z 306.377,A -85,B 0,C 180,E1 -9106.039,E2 -9106.039} C_VEL
LIN {X 0,Y 438.717,Z 293.283,A -85,B 0,C 180,E1 -9106.512,E2 -9106.512} C_VEL
LIN {X 0,Y 438.991,Z 283.583,A -85,B 0,C 180,E1 -9110.132,E2 -9110.132} C_VEL
LIN {X 0,Y 439.307,Z 274.647,A -85,B 0,C 180,E1 -9113.574,E2 -9113.574} C_VEL
LIN {X 0,Y 439.666,Z 267.038,A -85,B 0,C 180,E1 -9116.587,E2 -9116.587} C_VEL
LIN {X 0,Y 440.13,Z 259.588,A -85,B 0,C 180,E1 -9119.669,E2 -9119.669} C_VEL
LIN {X 0,Y 440.735,Z 252.273,A -85,B 0,C 180,E1 -9122.83,E2 -9122.83} C_VEL
LIN {X 0,Y 441.154,Z 246.046,A -85,B 0,C 180,E1 -9125.66,E2 -9125.66} C_VEL
LIN {X 0,Y 440.98,Z 242.765,A -85,B 0,C 180,E1 -9127.272,E2 -9127.272} C_VEL
LIN {X 0,Y 440.109,Z 237.693,A -85,B 0,C 180,E1 -9129.958,E2 -9129.958} C_VEL
LIN {X 0,Y 439.399,Z 233.756,A -85,B 0,C 180,E1 -9132.203,E2 -9132.203} C_VEL
LIN {X 0,Y 439.399,Z 233.753,A -85,B 0,C 180,E1 -9135.269,E2 -9135.269} C_VEL
LIN {X 0,Y 439.387,Z 233.756,A -85,B 0,C 180,E1 -9138.742,E2 -9138.742} C_VEL
LIN {X 0,Y 439.381,Z 233.756,A -85,B 0,C 180,E1 -9141.605,E2 -9141.605} C_VEL
LIN {X 0,Y 439.399,Z 233.754,A -85,B 0,C 180,E1 -9144.843,E2 -9144.843} C_VEL
LIN {X 0,Y 439.371,Z 233.757,A -85,B 0,C 180,E1 -9148.138,E2 -9148.138} C_VEL
LIN {X 0,Y 439.43,Z 233.75,A -85,B 0,C 180,E1 -9151.597,E2 -9151.597} C_VEL
LIN {X 0,Y 439.394,Z 233.755,A -85,B 0,C 180,E1 -9154.413,E2 -9154.413} C_VEL
LIN {X 0,Y 439.36,Z 233.757,A -85,B 0,C 180,E1 -9157.423,E2 -9157.423} C_VEL
LIN {X 0,Y 439.438,Z 233.748,A -85,B 0,C 180,E1 -9160.661,E2 -9160.661} C_VEL
LIN {X 0,Y 439.458,Z 233.745,A -85,B 0,C 180,E1 -9164.223,E2 -9164.223} C_VEL
LIN {X 0,Y 439.503,Z 233.741,A -85,B 0,C 180,E1 -9168.001,E2 -9168.001} C_VEL
LIN {X 0,Y 439.543,Z 233.736,A -85,B 0,C 180,E1 -9171.725,E2 -9171.725} C_VEL
LIN {X 0,Y 439.616,Z 233.725,A -85,B 0,C 180,E1 -9174.494,E2 -9174.494} C_VEL
LIN {X 0,Y 439.63,Z 233.725,A -85,B 0,C 180,E1 -9178.166,E2 -9178.166} C_VEL
LIN {X 0,Y 439.758,Z 233.709,A -85,B 0,C 180,E1 -9179.999,E2 -9179.999} C_VEL
LIN {X 0,Y 439.65,Z 233.722,A -85,B 0,C 180,E1 -9182.747,E2 -9182.747} C_VEL
LIN {X 0,Y 439.611,Z 233.728,A -85,B 0,C 180,E1 -9186.424,E2 -9186.424} C_VEL
LIN {X 0,Y 439.495,Z 233.741,A -85,B 0,C 180,E1 -9189.2,E2 -9189.2} C_VEL
LIN {X 0,Y 439.495,Z 233.742,A -85,B 0,C 180,E1 -9192.726,E2 -9192.726} C_VEL
LIN {X 0,Y 439.44,Z 233.752,A -85,B 0,C 180,E1 -9196.349,E2 -9196.349} C_VEL
LIN {X 0,Y 439.111,Z 233.792,A -85,B 0,C 180,E1 -9199.638,E2 -9199.638} C_VEL
LIN {X 0,Y 439.088,Z 235.3,A -85,B 0,C 180,E1 -9201.599,E2 -9201.599} C_VEL
LIN {X 0,Y 438.944,Z 238.176,A -85,B 0,C 180,E1 -9204.599,E2 -9204.599} C_VEL
LIN {X 0,Y 438.813,Z 241.213,A -85,B 0,C 180,E1 -9207.673,E2 -9207.673} C_VEL
LIN {X 0,Y 438.752,Z 244.376,A -85,B 0,C 180,E1 -9210.834,E2 -9210.834} C_VEL
LIN {X 0,Y 438.617,Z 247.706,A -85,B 0,C 180,E1 -9214.109,E2 -9214.109} C_VEL
LIN {X 0,Y 438.609,Z 250.505,A -85,B 0,C 180,E1 -9216.638,E2 -9216.638} C_VEL
LIN {X 0,Y 442.068,Z 264.079,A -85,B 0,C 180,E1 -9217.234,E2 -9217.234} C_VEL
LIN {X 0,Y 443.035,Z 269.589,A -85,B 0,C 180,E1 -9217.519,E2 -9217.519} C_VEL
LIN {X 0,Y 442.53,Z 281.874,A -85,B 0,C 180,E1 -9218.188,E2 -9218.188} C_VEL
LIN {X 0,Y 441.895,Z 293.488,A -85,B 0,C 180,E1 -9219.024,E2 -9219.024} C_VEL
LIN {X 0,Y 441.287,Z 304.645,A -85,B 0,C 180,E1 -9220.045,E2 -9220.045} C_VEL
LIN {X 0,Y 440.703,Z 314.117,A -85,B 0,C 180,E1 -9221.121,E2 -9221.121} C_VEL
LIN {X 0,Y 440.06,Z 323.223,A -85,B 0,C 180,E1 -9222.401,E2 -9222.401} C_VEL
LIN {X 0,Y 439.609,Z 330.719,A -85,B 0,C 180,E1 -9223.7,E2 -9223.7} C_VEL
LIN {X 0,Y 439.157,Z 337.839,A -85,B 0,C 180,E1 -9225.241,E2 -9225.241} C_VEL
LIN {X 0,Y 438.862,Z 342.374,A -85,B 0,C 180,E1 -9226.481,E2 -9226.481} C_VEL
LIN {X 0,Y 438.645,Z 345.934,A -85,B 0,C 180,E1 -9227.708,E2 -9227.708} C_VEL
LIN {X 0,Y 438.497,Z 348.658,A -85,B 0,C 180,E1 -9228.92,E2 -9228.92} C_VEL
LIN {X 0,Y 438.35,Z 350.876,A -85,B 0,C 180,E1 -9230.313,E2 -9230.313} C_VEL
LIN {X 0,Y 438.246,Z 352.204,A -85,B 0,C 180,E1 -9231.791,E2 -9231.791} C_VEL
LIN {X 0,Y 438.228,Z 352.443,A -85,B 0,C 180,E1 -9233.604,E2 -9233.604} C_VEL
LIN {X 0,Y 438.279,Z 351.69,A -85,B 0,C 180,E1 -9234.862,E2 -9234.862} C_VEL
LIN {X 0,Y 438.376,Z 349.652,A -85,B 0,C 180,E1 -9236.473,E2 -9236.473} C_VEL
LIN {X 0,Y 438.608,Z 346.234,A -85,B 0,C 180,E1 -9238.125,E2 -9238.125} C_VEL
LIN {X 0,Y 438.859,Z 341.033,A -85,B 0,C 180,E1 -9239.852,E2 -9239.852} C_VEL
LIN {X 0,Y 439.203,Z 335.23,A -85,B 0,C 180,E1 -9241.312,E2 -9241.312} C_VEL
LIN {X 0,Y 439.62,Z 328.628,A -85,B 0,C 180,E1 -9242.639,E2 -9242.639} C_VEL
LIN {X 0,Y 440.141,Z 320.53,A -85,B 0,C 180,E1 -9243.954,E2 -9243.954} C_VEL
LIN {X 0,Y 440.726,Z 311.133,A -85,B 0,C 180,E1 -9245.188,E2 -9245.188} C_VEL
LIN {X 0,Y 441.319,Z 300.766,A -85,B 0,C 180,E1 -9246.291,E2 -9246.291} C_VEL
LIN {X 0,Y 441.856,Z 290.589,A -85,B 0,C 180,E1 -9247.164,E2 -9247.164} C_VEL
LIN {X 0,Y 442.354,Z 278.908,A -85,B 0,C 180,E1 -9247.955,E2 -9247.955} C_VEL
LIN {X 0,Y 442.783,Z 267.896,A -85,B 0,C 180,E1 -9248.528,E2 -9248.528} C_VEL
LIN {X 0,Y 439.982,Z 255.292,A -85,B 0,C 180,E1 -9249.121,E2 -9249.121} C_VEL
LIN {X 0,Y 438.565,Z 249.342,A -85,B 0,C 180,E1 -9249.358,E2 -9249.358} C_VEL
LIN {X 0,Y 438.595,Z 246.153,A -85,B 0,C 180,E1 -9252.321,E2 -9252.321} C_VEL
LIN {X 0,Y 438.663,Z 243.121,A -85,B 0,C 180,E1 -9255.148,E2 -9255.148} C_VEL
LIN {X 0,Y 438.672,Z 241.932,A -85,B 0,C 180,E1 -9256.279,E2 -9256.279} C_VEL
LIN {X 0,Y 437.995,Z 241.201,A -85,B 0,C 180,E1 -9257.04,E2 -9257.04} C_VEL
LIN {X 0,Y 435.143,Z 240.202,A -85,B 0,C 180,E1 -9258.28,E2 -9258.28} C_VEL
LIN {X 0,Y 432.767,Z 239.4,A -85,B 0,C 180,E1 -9259.281,E2 -9259.281} C_VEL
LIN {X 0,Y 431.788,Z 238.711,A -85,B 0,C 180,E1 -9260.053,E2 -9260.053} C_VEL
LIN {X 0,Y 431.73,Z 238.44,A -85,B 0,C 180,E1 -9260.314,E2 -9260.314} C_VEL
LIN {X 0,Y 431.888,Z 235.217,A -85,B 0,C 180,E1 -9263.46,E2 -9263.46} C_VEL
LIN {X 0,Y 431.977,Z 234.678,A -85,B 0,C 180,E1 -9264.399,E2 -9264.399} C_VEL
LIN {X 0,Y 432.518,Z 234.609,A -85,B 0,C 180,E1 -9268.139,E2 -9268.139} C_VEL
LIN {X 0,Y 432.717,Z 234.584,A -85,B 0,C 180,E1 -9270.001,E2 -9270.001} C_VEL
LIN {X 0,Y 432.593,Z 234.6,A -85,B 0,C 180,E1 -9272.795,E2 -9272.795} C_VEL
LIN {X 0,Y 432.559,Z 234.604,A -85,B 0,C 180,E1 -9276.531,E2 -9276.531} C_VEL
LIN {X 0,Y 432.433,Z 234.622,A -85,B 0,C 180,E1 -9279.354,E2 -9279.354} C_VEL
LIN {X 0,Y 432.432,Z 234.621,A -85,B 0,C 180,E1 -9282.813,E2 -9282.813} C_VEL
LIN {X 0,Y 432.4,Z 234.623,A -85,B 0,C 180,E1 -9286.48,E2 -9286.48} C_VEL
LIN {X 0,Y 432.368,Z 234.627,A -85,B 0,C 180,E1 -9289.96,E2 -9289.96} C_VEL
LIN {X 0,Y 432.314,Z 234.636,A -85,B 0,C 180,E1 -9292.965,E2 -9292.965} C_VEL
LIN {X 0,Y 432.354,Z 234.629,A -85,B 0,C 180,E1 -9296.034,E2 -9296.034} C_VEL
LIN {X 0,Y 432.333,Z 234.633,A -85,B 0,C 180,E1 -9299.189,E2 -9299.189} C_VEL
LIN {X 0,Y 432.314,Z 234.635,A -85,B 0,C 180,E1 -9302.445,E2 -9302.445} C_VEL
LIN {X 0,Y 432.337,Z 234.63,A -85,B 0,C 180,E1 -9305.634,E2 -9305.634} C_VEL
LIN {X 0,Y 432.352,Z 234.632,A -85,B 0,C 180,E1 -9308.72,E2 -9308.72} C_VEL
LIN {X 0,Y 432.367,Z 234.627,A -85,B 0,C 180,E1 -9311.794,E2 -9311.794} C_VEL
LIN {X 0,Y 432.373,Z 234.63,A -85,B 0,C 180,E1 -9314.343,E2 -9314.343} C_VEL
LIN {X 0,Y 432.362,Z 234.63,A -85,B 0,C 180,E1 -9318.395,E2 -9318.395} C_VEL
LIN {X 0,Y 432.35,Z 234.629,A -85,B 0,C 180,E1 -9321.854,E2 -9321.854} C_VEL
LIN {X 0,Y 432.338,Z 234.631,A -85,B 0,C 180,E1 -9325.325,E2 -9325.325} C_VEL
LIN {X 0,Y 432.32,Z 234.636,A -85,B 0,C 180,E1 -9328.656,E2 -9328.656} C_VEL
LIN {X 0,Y 432.381,Z 234.627,A -85,B 0,C 180,E1 -9331.879,E2 -9331.879} C_VEL
LIN {X 0,Y 432.347,Z 234.629,A -85,B 0,C 180,E1 -9335,E2 -9335} C_VEL
LIN {X 0,Y 432.359,Z 234.631,A -85,B 0,C 180,E1 -9338.048,E2 -9338.048} C_VEL
LIN {X 0,Y 432.389,Z 234.624,A -85,B 0,C 180,E1 -9341.032,E2 -9341.032} C_VEL
LIN {X 0,Y 432.434,Z 234.623,A -85,B 0,C 180,E1 -9343.963,E2 -9343.963} C_VEL
LIN {X 0,Y 432.485,Z 234.615,A -85,B 0,C 180,E1 -9347.806,E2 -9347.806} C_VEL
LIN {X 0,Y 432.469,Z 234.616,A -85,B 0,C 180,E1 -9351.591,E2 -9351.591} C_VEL
LIN {X 0,Y 432.601,Z 234.599,A -85,B 0,C 180,E1 -9354.408,E2 -9354.408} C_VEL
LIN {X 0,Y 432.61,Z 234.599,A -85,B 0,C 180,E1 -9358.14,E2 -9358.14} C_VEL
LIN {X 0,Y 432.739,Z 234.583,A -85,B 0,C 180,E1 -9360.001,E2 -9360.001} C_VEL
LIN {X 0,Y 432.591,Z 234.598,A -85,B 0,C 180,E1 -9362.795,E2 -9362.795} C_VEL
LIN {X 0,Y 432.598,Z 234.602,A -85,B 0,C 180,E1 -9365.595,E2 -9365.595} C_VEL
LIN {X 0,Y 432.472,Z 234.614,A -85,B 0,C 180,E1 -9368.411,E2 -9368.411} C_VEL
LIN {X 0,Y 432.468,Z 234.616,A -85,B 0,C 180,E1 -9372.198,E2 -9372.198} C_VEL
LIN {X 0,Y 432.439,Z 234.618,A -85,B 0,C 180,E1 -9376.04,E2 -9376.04} C_VEL
LIN {X 0,Y 432.396,Z 234.627,A -85,B 0,C 180,E1 -9379.486,E2 -9379.486} C_VEL
LIN {X 0,Y 432.326,Z 234.635,A -85,B 0,C 180,E1 -9382.965,E2 -9382.965} C_VEL
LIN {X 0,Y 432.359,Z 234.629,A -85,B 0,C 180,E1 -9386.034,E2 -9386.034} C_VEL
LIN {X 0,Y 432.352,Z 234.632,A -85,B 0,C 180,E1 -9389.188,E2 -9389.188} C_VEL
LIN {X 0,Y 432.332,Z 234.632,A -85,B 0,C 180,E1 -9392.443,E2 -9392.443} C_VEL
LIN {X 0,Y 432.352,Z 234.63,A -85,B 0,C 180,E1 -9395.632,E2 -9395.632} C_VEL
LIN {X 0,Y 432.343,Z 234.632,A -85,B 0,C 180,E1 -9398.713,E2 -9398.713} C_VEL
LIN {X 0,Y 432.342,Z 234.631,A -85,B 0,C 180,E1 -9401.797,E2 -9401.797} C_VEL
LIN {X 0,Y 432.343,Z 234.631,A -85,B 0,C 180,E1 -9404.347,E2 -9404.347} C_VEL
LIN {X 0,Y 432.373,Z 234.626,A -85,B 0,C 180,E1 -9408.05,E2 -9408.05} C_VEL
LIN {X 0,Y 433.25,Z 239.702,A -85,B 0,C 180,E1 -9410.754,E2 -9410.754} C_VEL
LIN {X 0,Y 434.075,Z 244.723,A -85,B 0,C 180,E1 -9413.197,E2 -9413.197} C_VEL
LIN {X 0,Y 434.13,Z 248.485,A -85,B 0,C 180,E1 -9414.92,E2 -9414.92} C_VEL
LIN {X 0,Y 433.661,Z 254.737,A -85,B 0,C 180,E1 -9417.668,E2 -9417.668} C_VEL
LIN {X 0,Y 433.048,Z 263.109,A -85,B 0,C 180,E1 -9421.209,E2 -9421.209} C_VEL
LIN {X 0,Y 432.557,Z 271.155,A -85,B 0,C 180,E1 -9424.496,E2 -9424.496} C_VEL
LIN {X 0,Y 432.175,Z 278.783,A -85,B 0,C 180,E1 -9427.532,E2 -9427.532} C_VEL
LIN {X 0,Y 431.824,Z 287.691,A -85,B 0,C 180,E1 -9431.003,E2 -9431.003} C_VEL
LIN {X 0,Y 431.678,Z 294.113,A -85,B 0,C 180,E1 -9433.377,E2 -9433.377} C_VEL
LIN {X 0,Y 433.679,Z 307.614,A -85,B 0,C 180,E1 -9433.839,E2 -9433.839} C_VEL
LIN {X 0,Y 435.185,Z 320.857,A -85,B 0,C 180,E1 -9434.485,E2 -9434.485} C_VEL
LIN {X 0,Y 434.536,Z 333.497,A -85,B 0,C 180,E1 -9435.241,E2 -9435.241} C_VEL
LIN {X 0,Y 433.851,Z 345.104,A -85,B 0,C 180,E1 -9436.152,E2 -9436.152} C_VEL
LIN {X 0,Y 433.195,Z 355.979,A -85,B 0,C 180,E1 -9437.229,E2 -9437.229} C_VEL
LIN {X 0,Y 432.697,Z 364.678,A -85,B 0,C 180,E1 -9438.285,E2 -9438.285} C_VEL
LIN {X 0,Y 432.185,Z 372.694,A -85,B 0,C 180,E1 -9439.458,E2 -9439.458} C_VEL
LIN {X 0,Y 431.753,Z 380.55,A -85,B 0,C 180,E1 -9440.867,E2 -9440.867} C_VEL
LIN {X 0,Y 431.467,Z 387.751,A -85,B 0,C 180,E1 -9442.512,E2 -9442.512} C_VEL
LIN {X 0,Y 431.293,Z 392.843,A -85,B 0,C 180,E1 -9444.014,E2 -9444.014} C_VEL
LIN {X 0,Y 431.285,Z 396.225,A -85,B 0,C 180,E1 -9445.326,E2 -9445.326} C_VEL
LIN {X 0,Y 431.232,Z 398.117,A -85,B 0,C 180,E1 -9446.261,E2 -9446.261} C_VEL
LIN {X 0,Y 431.32,Z 399.549,A -85,B 0,C 180,E1 -9447.197,E2 -9447.197} C_VEL
LIN {X 0,Y 431.279,Z 401.165,A -85,B 0,C 180,E1 -9449.065,E2 -9449.065} C_VEL
LIN {X 0,Y 431.285,Z 401.385,A -85,B 0,C 180,E1 -9449.999,E2 -9449.999} C_VEL
LIN {X 0,Y 431.264,Z 401.168,A -85,B 0,C 180,E1 -9450.933,E2 -9450.933} C_VEL
LIN {X 0,Y 431.319,Z 399.53,A -85,B 0,C 180,E1 -9452.801,E2 -9452.801} C_VEL
LIN {X 0,Y 431.23,Z 398.106,A -85,B 0,C 180,E1 -9453.737,E2 -9453.737} C_VEL
LIN {X 0,Y 431.322,Z 395.126,A -85,B 0,C 180,E1 -9455.141,E2 -9455.141} C_VEL
LIN {X 0,Y 431.379,Z 391.098,A -85,B 0,C 180,E1 -9456.548,E2 -9456.548} C_VEL
LIN {X 0,Y 431.586,Z 384.924,A -85,B 0,C 180,E1 -9458.191,E2 -9458.191} C_VEL
LIN {X 0,Y 431.883,Z 378.182,A -85,B 0,C 180,E1 -9459.601,E2 -9459.601} C_VEL
LIN {X 0,Y 432.357,Z 369.835,A -85,B 0,C 180,E1 -9461.01,E2 -9461.01} C_VEL
LIN {X 0,Y 432.958,Z 361.315,A -85,B 0,C 180,E1 -9462.181,E2 -9462.181} C_VEL
LIN {X 0,Y 433.522,Z 350.988,A -85,B 0,C 180,E1 -9463.338,E2 -9463.338} C_VEL
LIN {X 0,Y 434.157,Z 340.465,A -85,B 0,C 180,E1 -9464.291,E2 -9464.291} C_VEL
LIN {X 0,Y 434.906,Z 329.192,A -85,B 0,C 180,E1 -9465.103,E2 -9465.103} C_VEL
LIN {X 0,Y 435.185,Z 320.048,A -85,B 0,C 180,E1 -9465.633,E2 -9465.633} C_VEL
LIN {X 0,Y 433.82,Z 306.954,A -85,B 0,C 180,E1 -9466.277,E2 -9466.277} C_VEL
LIN {X 0,Y 431.723,Z 293.749,A -85,B 0,C 180,E1 -9466.754,E2 -9466.754} C_VEL
LIN {X 0,Y 431.646,Z 292.919,A -85,B 0,C 180,E1 -9466.776,E2 -9466.776} C_VEL
LIN {X 0,Y 431.935,Z 283.238,A -85,B 0,C 180,E1 -9470.476,E2 -9470.476} C_VEL
LIN {X 0,Y 432.224,Z 275.608,A -85,B 0,C 180,E1 -9473.475,E2 -9473.475} C_VEL
LIN {X 0,Y 432.631,Z 267.654,A -85,B 0,C 180,E1 -9476.687,E2 -9476.687} C_VEL
LIN {X 0,Y 433.158,Z 259.351,A -85,B 0,C 180,E1 -9480.196,E2 -9480.196} C_VEL
LIN {X 0,Y 433.83,Z 252.115,A -85,B 0,C 180,E1 -9483.42,E2 -9483.42} C_VEL
LIN {X 0,Y 434.203,Z 246.697,A -85,B 0,C 180,E1 -9485.971,E2 -9485.971} C_VEL
LIN {X 0,Y 433.81,Z 242.708,A -85,B 0,C 180,E1 -9487.996,E2 -9487.996} C_VEL
LIN {X 0,Y 432.844,Z 237.16,A -85,B 0,C 180,E1 -9491.059,E2 -9491.059} C_VEL
LIN {X 0,Y 432.356,Z 234.631,A -85,B 0,C 180,E1 -9492.579,E2 -9492.579} C_VEL
LIN {X 0,Y 432.332,Z 234.635,A -85,B 0,C 180,E1 -9495.663,E2 -9495.663} C_VEL
LIN {X 0,Y 432.332,Z 234.634,A -85,B 0,C 180,E1 -9498.397,E2 -9498.397} C_VEL
LIN {X 0,Y 432.344,Z 234.633,A -85,B 0,C 180,E1 -9501.85,E2 -9501.85} C_VEL
LIN {X 0,Y 432.339,Z 234.634,A -85,B 0,C 180,E1 -9505.322,E2 -9505.322} C_VEL
LIN {X 0,Y 432.319,Z 234.635,A -85,B 0,C 180,E1 -9508.653,E2 -9508.653} C_VEL
LIN {X 0,Y 432.38,Z 234.627,A -85,B 0,C 180,E1 -9511.875,E2 -9511.875} C_VEL
LIN {X 0,Y 432.343,Z 234.633,A -85,B 0,C 180,E1 -9514.997,E2 -9514.997} C_VEL
LIN {X 0,Y 432.354,Z 234.632,A -85,B 0,C 180,E1 -9518.044,E2 -9518.044} C_VEL
LIN {X 0,Y 432.383,Z 234.627,A -85,B 0,C 180,E1 -9521.028,E2 -9521.028} C_VEL
LIN {X 0,Y 432.427,Z 234.621,A -85,B 0,C 180,E1 -9523.96,E2 -9523.96} C_VEL
LIN {X 0,Y 432.476,Z 234.615,A -85,B 0,C 180,E1 -9527.803,E2 -9527.803} C_VEL
LIN {X 0,Y 432.487,Z 234.615,A -85,B 0,C 180,E1 -9531.589,E2 -9531.589} C_VEL
LIN {X 0,Y 432.593,Z 234.6,A -85,B 0,C 180,E1 -9534.405,E2 -9534.405} C_VEL
LIN {X 0,Y 432.6,Z 234.6,A -85,B 0,C 180,E1 -9538.137,E2 -9538.137} C_VEL
LIN {X 0,Y 432.727,Z 234.584,A -85,B 0,C 180,E1 -9539.999,E2 -9539.999} C_VEL
LIN {X 0,Y 432.6,Z 234.601,A -85,B 0,C 180,E1 -9542.792,E2 -9542.792} C_VEL
LIN {X 0,Y 432.565,Z 234.604,A -85,B 0,C 180,E1 -9546.529,E2 -9546.529} C_VEL
LIN {X 0,Y 432.438,Z 234.62,A -85,B 0,C 180,E1 -9549.352,E2 -9549.352} C_VEL
LIN {X 0,Y 432.436,Z 234.621,A -85,B 0,C 180,E1 -9552.811,E2 -9552.811} C_VEL
LIN {X 0,Y 432.387,Z 234.631,A -85,B 0,C 180,E1 -9556.471,E2 -9556.471} C_VEL
LIN {X 0,Y 432.105,Z 234.664,A -85,B 0,C 180,E1 -9559.382,E2 -9559.382} C_VEL
LIN {X 0,Y 432.023,Z 234.675,A -85,B 0,C 180,E1 -9559.974,E2 -9559.974} C_VEL
LIN {X 0,Y 431.942,Z 237.514,A -85,B 0,C 180,E1 -9562.983,E2 -9562.983} C_VEL
LIN {X 0,Y 431.829,Z 240.443,A -85,B 0,C 180,E1 -9566.065,E2 -9566.065} C_VEL
LIN {X 0,Y 431.728,Z 243.571,A -85,B 0,C 180,E1 -9569.231,E2 -9569.231} C_VEL
LIN {X 0,Y 431.615,Z 246.829,A -85,B 0,C 180,E1 -9572.501,E2 -9572.501} C_VEL
LIN {X 0,Y 431.506,Z 250.283,A -85,B 0,C 180,E1 -9575.895,E2 -9575.895} C_VEL
LIN {X 0,Y 431.525,Z 250.728,A -85,B 0,C 180,E1 -9576.326,E2 -9576.326} C_VEL
LIN {X 0,Y 435.141,Z 264.908,A -85,B 0,C 180,E1 -9576.979,E2 -9576.979} C_VEL
LIN {X 0,Y 436.241,Z 270.182,A -85,B 0,C 180,E1 -9577.268,E2 -9577.268} C_VEL
LIN {X 0,Y 435.714,Z 282.155,A -85,B 0,C 180,E1 -9577.931,E2 -9577.931} C_VEL
LIN {X 0,Y 435.059,Z 293.453,A -85,B 0,C 180,E1 -9578.751,E2 -9578.751} C_VEL
LIN {X 0,Y 434.489,Z 303.903,A -85,B 0,C 180,E1 -9579.709,E2 -9579.709} C_VEL
LIN {X 0,Y 433.89,Z 313.396,A -85,B 0,C 180,E1 -9580.778,E2 -9580.778} C_VEL
LIN {X 0,Y 433.197,Z 322.767,A -85,B 0,C 180,E1 -9582.08,E2 -9582.08} C_VEL
LIN {X 0,Y 432.673,Z 330.294,A -85,B 0,C 180,E1 -9583.376,E2 -9583.376} C_VEL
LIN {X 0,Y 432.274,Z 336.397,A -85,B 0,C 180,E1 -9584.661,E2 -9584.661} C_VEL
LIN {X 0,Y 431.852,Z 342.545,A -85,B 0,C 180,E1 -9586.294,E2 -9586.294} C_VEL
LIN {X 0,Y 431.584,Z 346.321,A -85,B 0,C 180,E1 -9587.602,E2 -9587.602} C_VEL
LIN {X 0,Y 431.36,Z 349.961,A -85,B 0,C 180,E1 -9589.331,E2 -9589.331} C_VEL
LIN {X 0,Y 431.241,Z 351.609,A -85,B 0,C 180,E1 -9590.538,E2 -9590.538} C_VEL
LIN {X 0,Y 431.166,Z 352.592,A -85,B 0,C 180,E1 -9591.729,E2 -9591.729} C_VEL
LIN {X 0,Y 431.17,Z 352.949,A -85,B 0,C 180,E1 -9593.002,E2 -9593.002} C_VEL
LIN {X 0,Y 431.17,Z 352.348,A -85,B 0,C 180,E1 -9594.583,E2 -9594.583} C_VEL
LIN {X 0,Y 431.28,Z 350.298,A -85,B 0,C 180,E1 -9596.356,E2 -9596.356} C_VEL
LIN {X 0,Y 431.505,Z 347.364,A -85,B 0,C 180,E1 -9597.876,E2 -9597.876} C_VEL
LIN {X 0,Y 431.779,Z 342.574,A -85,B 0,C 180,E1 -9599.614,E2 -9599.614} C_VEL
LIN {X 0,Y 432.138,Z 336.839,A -85,B 0,C 180,E1 -9601.148,E2 -9601.148} C_VEL
LIN {X 0,Y 432.574,Z 329.545,A -85,B 0,C 180,E1 -9602.68,E2 -9602.68} C_VEL
LIN {X 0,Y 433.127,Z 321.586,A -85,B 0,C 180,E1 -9604.018,E2 -9604.018} C_VEL
LIN {X 0,Y 433.652,Z 313.216,A -85,B 0,C 180,E1 -9605.166,E2 -9605.166} C_VEL
LIN {X 0,Y 434.276,Z 303.423,A -85,B 0,C 180,E1 -9606.263,E2 -9606.263} C_VEL
LIN {X 0,Y 434.91,Z 291.844,A -85,B 0,C 180,E1 -9607.307,E2 -9607.307} C_VEL
LIN {X 0,Y 435.463,Z 279.823,A -85,B 0,C 180,E1 -9608.149,E2 -9608.149} C_VEL
LIN {X 0,Y 435.917,Z 268.96,A -85,B 0,C 180,E1 -9608.732,E2 -9608.732} C_VEL
LIN {X 0,Y 432.997,Z 256.079,A -85,B 0,C 180,E1 -9609.36,E2 -9609.36} C_VEL
LIN {X 0,Y 431.489,Z 249.697,A -85,B 0,C 180,E1 -9609.627,E2 -9609.627} C_VEL
LIN {X 0,Y 431.516,Z 247.171,A -85,B 0,C 180,E1 -9611.975,E2 -9611.975} C_VEL
LIN {X 0,Y 431.616,Z 244.067,A -85,B 0,C 180,E1 -9614.9,E2 -9614.9} C_VEL
LIN {X 0,Y 431.727,Z 241.057,A -85,B 0,C 180,E1 -9617.783,E2 -9617.783} C_VEL
LIN {X 0,Y 431.73,Z 238.44,A -85,B 0,C 180,E1 -9620.314,E2 -9620.314} C_VEL
LIN {X 0,Y 431.129,Z 237.722,A -85,B 0,C 180,E1 -9621.087,E2 -9621.087} C_VEL
LIN {X 0,Y 428.341,Z 236.719,A -85,B 0,C 180,E1 -9622.349,E2 -9622.349} C_VEL
LIN {X 0,Y 425.973,Z 235.944,A -85,B 0,C 180,E1 -9623.37,E2 -9623.37} C_VEL
LIN {X 0,Y 424.989,Z 235.587,A -85,B 0,C 180,E1 -9624.159,E2 -9624.159} C_VEL
LIN {X 0,Y 424.928,Z 235.555,A -85,B 0,C 180,E1 -9624.427,E2 -9624.427} C_VEL
LIN {X 0,Y 425.48,Z 235.486,A -85,B 0,C 180,E1 -9628.108,E2 -9628.108} C_VEL
LIN {X 0,Y 425.687,Z 235.46,A -85,B 0,C 180,E1 -9630.001,E2 -9630.001} C_VEL
LIN {X 0,Y 425.544,Z 235.478,A -85,B 0,C 180,E1 -9632.841,E2 -9632.841} C_VEL
LIN {X 0,Y 425.517,Z 235.481,A -85,B 0,C 180,E1 -9636.64,E2 -9636.64} C_VEL
LIN {X 0,Y 425.392,Z 235.499,A -85,B 0,C 180,E1 -9639.511,E2 -9639.511} C_VEL
LIN {X 0,Y 425.391,Z 235.498,A -85,B 0,C 180,E1 -9642.912,E2 -9642.912} C_VEL
LIN {X 0,Y 425.349,Z 235.502,A -85,B 0,C 180,E1 -9646.606,E2 -9646.606} C_VEL
LIN {X 0,Y 425.35,Z 235.502,A -85,B 0,C 180,E1 -9649.65,E2 -9649.65} C_VEL
LIN {X 0,Y 425.299,Z 235.509,A -85,B 0,C 180,E1 -9653.367,E2 -9653.367} C_VEL
LIN {X 0,Y 425.338,Z 235.506,A -85,B 0,C 180,E1 -9656.846,E2 -9656.846} C_VEL
LIN {X 0,Y 425.281,Z 235.509,A -85,B 0,C 180,E1 -9659.721,E2 -9659.721} C_VEL
LIN {X 0,Y 425.273,Z 235.513,A -85,B 0,C 180,E1 -9663.05,E2 -9663.05} C_VEL
LIN {X 0,Y 425.277,Z 235.51,A -85,B 0,C 180,E1 -9665.931,E2 -9665.931} C_VEL
LIN {X 0,Y 425.305,Z 235.509,A -85,B 0,C 180,E1 -9669.048,E2 -9669.048} C_VEL
LIN {X 0,Y 425.325,Z 235.507,A -85,B 0,C 180,E1 -9672.648,E2 -9672.648} C_VEL
LIN {X 0,Y 425.289,Z 235.509,A -85,B 0,C 180,E1 -9675.284,E2 -9675.284} C_VEL
LIN {X 0,Y 425.3,Z 235.511,A -85,B 0,C 180,E1 -9678.627,E2 -9678.627} C_VEL
LIN {X 0,Y 425.321,Z 235.505,A -85,B 0,C 180,E1 -9681.106,E2 -9681.106} C_VEL
LIN {X 0,Y 425.298,Z 235.51,A -85,B 0,C 180,E1 -9684.666,E2 -9684.666} C_VEL
LIN {X 0,Y 425.264,Z 235.515,A -85,B 0,C 180,E1 -9688.075,E2 -9688.075} C_VEL
LIN {X 0,Y 425.331,Z 235.504,A -85,B 0,C 180,E1 -9691.37,E2 -9691.37} C_VEL
LIN {X 0,Y 425.354,Z 235.501,A -85,B 0,C 180,E1 -9693.507,E2 -9693.507} C_VEL
LIN {X 0,Y 425.306,Z 235.509,A -85,B 0,C 180,E1 -9696.637,E2 -9696.637} C_VEL
LIN {X 0,Y 425.331,Z 235.506,A -85,B 0,C 180,E1 -9700.366,E2 -9700.366} C_VEL
LIN {X 0,Y 425.392,Z 235.498,A -85,B 0,C 180,E1 -9703.69,E2 -9703.69} C_VEL
LIN {X 0,Y 425.434,Z 235.493,A -85,B 0,C 180,E1 -9707.601,E2 -9707.601} C_VEL
LIN {X 0,Y 425.413,Z 235.495,A -85,B 0,C 180,E1 -9711.451,E2 -9711.451} C_VEL
LIN {X 0,Y 425.556,Z 235.476,A -85,B 0,C 180,E1 -9714.315,E2 -9714.315} C_VEL
LIN {X 0,Y 425.579,Z 235.475,A -85,B 0,C 180,E1 -9718.109,E2 -9718.109} C_VEL
LIN {X 0,Y 425.708,Z 235.459,A -85,B 0,C 180,E1 -9720.001,E2 -9720.001} C_VEL
LIN {X 0,Y 425.545,Z 235.476,A -85,B 0,C 180,E1 -9722.841,E2 -9722.841} C_VEL
LIN {X 0,Y 425.554,Z 235.479,A -85,B 0,C 180,E1 -9725.688,E2 -9725.688} C_VEL
LIN {X 0,Y 425.416,Z 235.492,A -85,B 0,C 180,E1 -9728.552,E2 -9728.552} C_VEL
LIN {X 0,Y 425.421,Z 235.492,A -85,B 0,C 180,E1 -9732.403,E2 -9732.403} C_VEL
LIN {X 0,Y 425.397,Z 235.494,A -85,B 0,C 180,E1 -9736.313,E2 -9736.313} C_VEL
LIN {X 0,Y 425.337,Z 235.505,A -85,B 0,C 180,E1 -9739.636,E2 -9739.636} C_VEL
LIN {X 0,Y 425.313,Z 235.508,A -85,B 0,C 180,E1 -9743.366,E2 -9743.366} C_VEL
LIN {X 0,Y 425.35,Z 235.503,A -85,B 0,C 180,E1 -9746.843,E2 -9746.843} C_VEL
LIN {X 0,Y 425.3,Z 235.508,A -85,B 0,C 180,E1 -9749.72,E2 -9749.72} C_VEL
LIN {X 0,Y 425.291,Z 235.512,A -85,B 0,C 180,E1 -9753.048,E2 -9753.048} C_VEL
LIN {X 0,Y 425.291,Z 235.508,A -85,B 0,C 180,E1 -9755.929,E2 -9755.929} C_VEL
LIN {X 0,Y 425.286,Z 235.512,A -85,B 0,C 180,E1 -9759.04,E2 -9759.04} C_VEL
LIN {X 0,Y 425.299,Z 235.509,A -85,B 0,C 180,E1 -9761.958,E2 -9761.958} C_VEL
LIN {X 0,Y 425.294,Z 235.508,A -85,B 0,C 180,E1 -9765.283,E2 -9765.283} C_VEL
LIN {X 0,Y 425.354,Z 235.598,A -85,B 0,C 180,E1 -9767.929,E2 -9767.929} C_VEL
LIN {X 0,Y 426.453,Z 241.975,A -85,B 0,C 180,E1 -9771.225,E2 -9771.225} C_VEL
LIN {X 0,Y 427.147,Z 247.094,A -85,B 0,C 180,E1 -9773.729,E2 -9773.729} C_VEL
LIN {X 0,Y 426.944,Z 251.97,A -85,B 0,C 180,E1 -9775.965,E2 -9775.965} C_VEL
LIN {X 0,Y 426.347,Z 258.888,A -85,B 0,C 180,E1 -9779.003,E2 -9779.003} C_VEL
LIN {X 0,Y 425.835,Z 265.791,A -85,B 0,C 180,E1 -9781.941,E2 -9781.941} C_VEL
LIN {X 0,Y 425.379,Z 273.962,A -85,B 0,C 180,E1 -9785.327,E2 -9785.327} C_VEL
LIN {X 0,Y 424.978,Z 282.252,A -85,B 0,C 180,E1 -9788.664,E2 -9788.664} C_VEL
LIN {X 0,Y 424.681,Z 289.858,A -85,B 0,C 180,E1 -9791.673,E2 -9791.673} C_VEL
LIN {X 0,Y 424.604,Z 293.474,A -85,B 0,C 180,E1 -9793.084,E2 -9793.084} C_VEL
LIN {X 0,Y 426.826,Z 308.646,A -85,B 0,C 180,E1 -9793.645,E2 -9793.645} C_VEL
LIN {X 0,Y 428.215,Z 321.302,A -85,B 0,C 180,E1 -9794.287,E2 -9794.287} C_VEL
LIN {X 0,Y 427.651,Z 332.883,A -85,B 0,C 180,E1 -9794.998,E2 -9794.998} C_VEL
LIN {X 0,Y 426.902,Z 344.802,A -85,B 0,C 180,E1 -9795.946,E2 -9795.946} C_VEL
LIN {X 0,Y 426.24,Z 355.45,A -85,B 0,C 180,E1 -9797.017,E2 -9797.017} C_VEL
LIN {X 0,Y 425.707,Z 364.17,A -85,B 0,C 180,E1 -9798.09,E2 -9798.09} C_VEL
LIN {X 0,Y 425.165,Z 372.205,A -85,B 0,C 180,E1 -9799.282,E2 -9799.282} C_VEL
LIN {X 0,Y 424.708,Z 380.086,A -85,B 0,C 180,E1 -9800.714,E2 -9800.714} C_VEL
LIN {X 0,Y 424.386,Z 387.3,A -85,B 0,C 180,E1 -9802.386,E2 -9802.386} C_VEL
LIN {X 0,Y 424.248,Z 391.756,A -85,B 0,C 180,E1 -9803.699,E2 -9803.699} C_VEL
LIN {X 0,Y 424.215,Z 395.8,A -85,B 0,C 180,E1 -9805.247,E2 -9805.247} C_VEL
LIN {X 0,Y 424.14,Z 397.695,A -85,B 0,C 180,E1 -9806.199,E2 -9806.199} C_VEL
LIN {X 0,Y 424.247,Z 399.137,A -85,B 0,C 180,E1 -9807.15,E2 -9807.15} C_VEL
LIN {X 0,Y 424.192,Z 400.761,A -85,B 0,C 180,E1 -9809.05,E2 -9809.05} C_VEL
LIN {X 0,Y 424.196,Z 400.984,A -85,B 0,C 180,E1 -9809.999,E2 -9809.999} C_VEL
LIN {X 0,Y 424.178,Z 400.774,A -85,B 0,C 180,E1 -9810.948,E2 -9810.948} C_VEL
LIN {X 0,Y 424.198,Z 400.155,A -85,B 0,C 180,E1 -9811.898,E2 -9811.898} C_VEL
LIN {X 0,Y 424.228,Z 399.142,A -85,B 0,C 180,E1 -9812.848,E2 -9812.848} C_VEL
LIN {X 0,Y 424.138,Z 397.72,A -85,B 0,C 180,E1 -9813.799,E2 -9813.799} C_VEL
LIN {X 0,Y 424.231,Z 394.744,A -85,B 0,C 180,E1 -9815.227,E2 -9815.227} C_VEL
LIN {X 0,Y 424.302,Z 390.721,A -85,B 0,C 180,E1 -9816.657,E2 -9816.657} C_VEL
LIN {X 0,Y 424.51,Z 384.556,A -85,B 0,C 180,E1 -9818.328,E2 -9818.328} C_VEL
LIN {X 0,Y 424.852,Z 377.822,A -85,B 0,C 180,E1 -9819.761,E2 -9819.761} C_VEL
LIN {X 0,Y 425.362,Z 369.483,A -85,B 0,C 180,E1 -9821.193,E2 -9821.193} C_VEL
LIN {X 0,Y 425.969,Z 360.976,A -85,B 0,C 180,E1 -9822.384,E2 -9822.384} C_VEL
LIN {X 0,Y 426.557,Z 350.611,A -85,B 0,C 180,E1 -9823.566,E2 -9823.566} C_VEL
LIN {X 0,Y 427.367,Z 338.749,A -85,B 0,C 180,E1 -9824.645,E2 -9824.645} C_VEL
LIN {X 0,Y 428.162,Z 327.116,A -85,B 0,C 180,E1 -9825.469,E2 -9825.469} C_VEL
LIN {X 0,Y 428.322,Z 321.003,A -85,B 0,C 180,E1 -9825.829,E2 -9825.829} C_VEL
LIN {X 0,Y 426.932,Z 307.451,A -85,B 0,C 180,E1 -9826.528,E2 -9826.528} C_VEL
LIN {X 0,Y 424.924,Z 294.65,A -85,B 0,C 180,E1 -9827.021,E2 -9827.021} C_VEL
LIN {X 0,Y 424.558,Z 292.435,A -85,B 0,C 180,E1 -9827.102,E2 -9827.102} C_VEL
LIN {X 0,Y 424.853,Z 284.19,A -85,B 0,C 180,E1 -9830.326,E2 -9830.326} C_VEL
LIN {X 0,Y 425.157,Z 276.578,A -85,B 0,C 180,E1 -9833.373,E2 -9833.373} C_VEL
LIN {X 0,Y 425.575,Z 269.076,A -85,B 0,C 180,E1 -9836.479,E2 -9836.479} C_VEL
LIN {X 0,Y 426.135,Z 260.418,A -85,B 0,C 180,E1 -9840.199,E2 -9840.199} C_VEL
LIN {X 0,Y 426.719,Z 254.361,A -85,B 0,C 180,E1 -9842.921,E2 -9842.921} C_VEL
LIN {X 0,Y 427.18,Z 248.495,A -85,B 0,C 180,E1 -9845.718,E2 -9845.718} C_VEL
LIN {X 0,Y 426.906,Z 244.438,A -85,B 0,C 180,E1 -9847.794,E2 -9847.794} C_VEL
LIN {X 0,Y 425.813,Z 238.194,A -85,B 0,C 180,E1 -9851.313,E2 -9851.313} C_VEL
LIN {X 0,Y 425.275,Z 235.513,A -85,B 0,C 180,E1 -9852.998,E2 -9852.998} C_VEL
LIN {X 0,Y 425.261,Z 235.516,A -85,B 0,C 180,E1 -9856.043,E2 -9856.043} C_VEL
LIN {X 0,Y 425.273,Z 235.514,A -85,B 0,C 180,E1 -9858.62,E2 -9858.62} C_VEL
LIN {X 0,Y 425.308,Z 235.51,A -85,B 0,C 180,E1 -9861.101,E2 -9861.101} C_VEL
LIN {X 0,Y 425.299,Z 235.511,A -85,B 0,C 180,E1 -9864.663,E2 -9864.663} C_VEL
LIN {X 0,Y 425.263,Z 235.515,A -85,B 0,C 180,E1 -9868.072,E2 -9868.072} C_VEL
LIN {X 0,Y 425.329,Z 235.508,A -85,B 0,C 180,E1 -9871.366,E2 -9871.366} C_VEL
LIN {X 0,Y 425.351,Z 235.504,A -85,B 0,C 180,E1 -9873.504,E2 -9873.504} C_VEL
LIN {X 0,Y 425.301,Z 235.51,A -85,B 0,C 180,E1 -9876.633,E2 -9876.633} C_VEL
LIN {X 0,Y 425.325,Z 235.507,A -85,B 0,C 180,E1 -9880.363,E2 -9880.363} C_VEL
LIN {X 0,Y 425.384,Z 235.5,A -85,B 0,C 180,E1 -9883.687,E2 -9883.687} C_VEL
LIN {X 0,Y 425.425,Z 235.494,A -85,B 0,C 180,E1 -9887.597,E2 -9887.597} C_VEL
LIN {X 0,Y 425.438,Z 235.493,A -85,B 0,C 180,E1 -9891.448,E2 -9891.448} C_VEL
LIN {X 0,Y 425.549,Z 235.478,A -85,B 0,C 180,E1 -9894.312,E2 -9894.312} C_VEL
LIN {X 0,Y 425.57,Z 235.476,A -85,B 0,C 180,E1 -9898.106,E2 -9898.106} C_VEL
LIN {X 0,Y 425.697,Z 235.46,A -85,B 0,C 180,E1 -9899.999,E2 -9899.999} C_VEL
LIN {X 0,Y 425.551,Z 235.479,A -85,B 0,C 180,E1 -9902.838,E2 -9902.838} C_VEL
LIN {X 0,Y 425.523,Z 235.481,A -85,B 0,C 180,E1 -9906.644,E2 -9906.644} C_VEL
LIN {X 0,Y 425.397,Z 235.498,A -85,B 0,C 180,E1 -9909.508,E2 -9909.508} C_VEL
LIN {X 0,Y 425.396,Z 235.499,A -85,B 0,C 180,E1 -9912.909,E2 -9912.909} C_VEL
LIN {X 0,Y 425.337,Z 235.51,A -85,B 0,C 180,E1 -9916.597,E2 -9916.597} C_VEL
LIN {X 0,Y 425.059,Z 235.542,A -85,B 0,C 180,E1 -9919.537,E2 -9919.537} C_VEL
LIN {X 0,Y 424.986,Z 235.892,A -85,B 0,C 180,E1 -9920.319,E2 -9920.319} C_VEL
LIN {X 0,Y 424.883,Z 238.77,A -85,B 0,C 180,E1 -9923.388,E2 -9923.388} C_VEL
LIN {X 0,Y 424.745,Z 241.904,A -85,B 0,C 180,E1 -9926.685,E2 -9926.685} C_VEL
LIN {X 0,Y 424.66,Z 244.885,A -85,B 0,C 180,E1 -9929.766,E2 -9929.766} C_VEL
LIN {X 0,Y 424.545,Z 248.204,A -85,B 0,C 180,E1 -9933.11,E2 -9933.11} C_VEL
LIN {X 0,Y 424.466,Z 251.128,A -85,B 0,C 180,E1 -9936.022,E2 -9936.022} C_VEL
LIN {X 0,Y 428.077,Z 264.833,A -85,B 0,C 180,E1 -9936.666,E2 -9936.666} C_VEL
LIN {X 0,Y 429.436,Z 271.625,A -85,B 0,C 180,E1 -9937.044,E2 -9937.044} C_VEL
LIN {X 0,Y 428.857,Z 283.602,A -85,B 0,C 180,E1 -9937.739,E2 -9937.739} C_VEL
LIN {X 0,Y 428.159,Z 294.885,A -85,B 0,C 180,E1 -9938.588,E2 -9938.588} C_VEL
LIN {X 0,Y 427.511,Z 305.671,A -85,B 0,C 180,E1 -9939.615,E2 -9939.615} C_VEL
LIN {X 0,Y 426.842,Z 315.389,A -85,B 0,C 180,E1 -9940.766,E2 -9940.766} C_VEL
LIN {X 0,Y 426.124,Z 324.393,A -85,B 0,C 180,E1 -9942.084,E2 -9942.084} C_VEL
LIN {X 0,Y 425.637,Z 331.729,A -85,B 0,C 180,E1 -9943.407,E2 -9943.407} C_VEL
LIN {X 0,Y 425.201,Z 337.625,A -85,B 0,C 180,E1 -9944.707,E2 -9944.707} C_VEL
LIN {X 0,Y 424.861,Z 342.365,A -85,B 0,C 180,E1 -9945.993,E2 -9945.993} C_VEL
LIN {X 0,Y 424.512,Z 347.357,A -85,B 0,C 180,E1 -9947.75,E2 -9947.75} C_VEL
LIN {X 0,Y 424.397,Z 349.026,A -85,B 0,C 180,E1 -9948.518,E2 -9948.518} C_VEL
LIN {X 0,Y 424.255,Z 351.108,A -85,B 0,C 180,E1 -9949.757,E2 -9949.757} C_VEL
LIN {X 0,Y 424.108,Z 352.63,A -85,B 0,C 180,E1 -9951.152,E2 -9951.152} C_VEL
LIN {X 0,Y 424.069,Z 353.315,A -85,B 0,C 180,E1 -9952.698,E2 -9952.698} C_VEL
LIN {X 0,Y 424.094,Z 352.782,A -85,B 0,C 180,E1 -9954.55,E2 -9954.55} C_VEL
LIN {X 0,Y 424.171,Z 351.37,A -85,B 0,C 180,E1 -9955.935,E2 -9955.935} C_VEL
LIN {X 0,Y 424.373,Z 348.47,A -85,B 0,C 180,E1 -9957.626,E2 -9957.626} C_VEL
LIN {X 0,Y 424.667,Z 343.972,A -85,B 0,C 180,E1 -9959.376,E2 -9959.376} C_VEL
LIN {X 0,Y 424.949,Z 339.244,A -85,B 0,C 180,E1 -9960.762,E2 -9960.762} C_VEL
LIN {X 0,Y 425.366,Z 333.178,A -85,B 0,C 180,E1 -9962.177,E2 -9962.177} C_VEL
LIN {X 0,Y 425.821,Z 325.976,A -85,B 0,C 180,E1 -9963.538,E2 -9963.538} C_VEL
LIN {X 0,Y 426.424,Z 317.347,A -85,B 0,C 180,E1 -9964.856,E2 -9964.856} C_VEL
LIN {X 0,Y 427.15,Z 307.229,A -85,B 0,C 180,E1 -9966.1,E2 -9966.1} C_VEL
LIN {X 0,Y 427.781,Z 296.203,A -85,B 0,C 180,E1 -9967.193,E2 -9967.193} C_VEL
LIN {X 0,Y 428.436,Z 284.641,A -85,B 0,C 180,E1 -9968.089,E2 -9968.089} C_VEL
LIN {X 0,Y 428.973,Z 272.594,A -85,B 0,C 180,E1 -9968.811,E2 -9968.811} C_VEL
LIN {X 0,Y 428.797,Z 269.192,A -85,B 0,C 180,E1 -9968.991,E2 -9968.991} C_VEL
LIN {X 0,Y 426.06,Z 256.761,A -85,B 0,C 180,E1 -9969.608,E2 -9969.608} C_VEL
LIN {X 0,Y 424.41,Z 250.084,A -85,B 0,C 180,E1 -9969.873,E2 -9969.873} C_VEL
LIN {X 0,Y 424.484,Z 247.109,A -85,B 0,C 180,E1 -9972.662,E2 -9972.662} C_VEL
LIN {X 0,Y 424.538,Z 244.015,A -85,B 0,C 180,E1 -9975.623,E2 -9975.623} C_VEL
LIN {X 0,Y 424.656,Z 240.977,A -85,B 0,C 180,E1 -9978.546,E2 -9978.546} C_VEL
LIN {X 0,Y 424.765,Z 238.029,A -85,B 0,C 180,E1 -9981.437,E2 -9981.437} C_VEL
LIN {X 0,Y 424.846,Z 236.084,A -85,B 0,C 180,E1 -9983.351,E2 -9983.351} C_VEL
LIN {X 0,Y 424.928,Z 235.555,A -85,B 0,C 180,E1 -9984.427,E2 -9984.427} C_VEL
LIN {X 0,Y 424.358,Z 235.629,A -85,B 0,C 180,E1 -9985.219,E2 -9985.219} C_VEL
LIN {X 0,Y 421.713,Z 235.955,A -85,B 0,C 180,E1 -9986.51,E2 -9986.51} C_VEL
LIN {X 0,Y 419.458,Z 236.239,A -85,B 0,C 180,E1 -9987.553,E2 -9987.553} C_VEL
LIN {X 0,Y 418.511,Z 236.353,A -85,B 0,C 180,E1 -9988.356,E2 -9988.356} C_VEL
LIN {X 0,Y 418.446,Z 236.361,A -85,B 0,C 180,E1 -9988.627,E2 -9988.627} C_VEL
LIN {X 0,Y 418.656,Z 236.335,A -85,B 0,C 180,E1 -9990.001,E2 -9990.001} C_VEL
LIN {X 0,Y 418.498,Z 236.356,A -85,B 0,C 180,E1 -9992.889,E2 -9992.889} C_VEL
LIN {X 0,Y 418.48,Z 236.359,A -85,B 0,C 180,E1 -9996.752,E2 -9996.752} C_VEL
LIN {X 0,Y 418.348,Z 236.374,A -85,B 0,C 180,E1 -9999.672,E2 -9999.672} C_VEL
LIN {X 0,Y 418.343,Z 236.377,A -85,B 0,C 180,E1 -10003.008,E2 -10003.008} C_VEL
LIN {X 0,Y 418.3,Z 236.381,A -85,B 0,C 180,E1 -10006.737,E2 -10006.737} C_VEL
LIN {X 0,Y 418.291,Z 236.381,A -85,B 0,C 180,E1 -10009.804,E2 -10009.804} C_VEL
LIN {X 0,Y 418.231,Z 236.391,A -85,B 0,C 180,E1 -10012.738,E2 -10012.738} C_VEL
LIN {X 0,Y 418.261,Z 236.384,A -85,B 0,C 180,E1 -10015.906,E2 -10015.906} C_VEL
LIN {X 0,Y 418.255,Z 236.387,A -85,B 0,C 180,E1 -10019.164,E2 -10019.164} C_VEL
LIN {X 0,Y 418.248,Z 236.389,A -85,B 0,C 180,E1 -10022.846,E2 -10022.846} C_VEL
LIN {X 0,Y 418.241,Z 236.388,A -85,B 0,C 180,E1 -10026.241,E2 -10026.241} C_VEL
LIN {X 0,Y 418.259,Z 236.384,A -85,B 0,C 180,E1 -10029.682,E2 -10029.682} C_VEL
LIN {X 0,Y 418.279,Z 236.384,A -85,B 0,C 180,E1 -10032.332,E2 -10032.332} C_VEL
LIN {X 0,Y 418.246,Z 236.387,A -85,B 0,C 180,E1 -10035.113,E2 -10035.113} C_VEL
LIN {X 0,Y 418.252,Z 236.386,A -85,B 0,C 180,E1 -10037.771,E2 -10037.771} C_VEL
LIN {X 0,Y 418.265,Z 236.387,A -85,B 0,C 180,E1 -10040.619,E2 -10040.619} C_VEL
LIN {X 0,Y 418.244,Z 236.388,A -85,B 0,C 180,E1 -10043.978,E2 -10043.978} C_VEL
LIN {X 0,Y 418.256,Z 236.384,A -85,B 0,C 180,E1 -10047.158,E2 -10047.158} C_VEL
LIN {X 0,Y 418.268,Z 236.384,A -85,B 0,C 180,E1 -10050.898,E2 -10050.898} C_VEL
LIN {X 0,Y 418.268,Z 236.386,A -85,B 0,C 180,E1 -10054.098,E2 -10054.098} C_VEL
LIN {X 0,Y 418.239,Z 236.387,A -85,B 0,C 180,E1 -10057.266,E2 -10057.266} C_VEL
LIN {X 0,Y 418.286,Z 236.384,A -85,B 0,C 180,E1 -10060.366,E2 -10060.366} C_VEL
LIN {X 0,Y 418.32,Z 236.377,A -85,B 0,C 180,E1 -10063.407,E2 -10063.407} C_VEL
LIN {X 0,Y 418.36,Z 236.371,A -85,B 0,C 180,E1 -10066.996,E2 -10066.996} C_VEL
LIN {X 0,Y 418.346,Z 236.376,A -85,B 0,C 180,E1 -10070.33,E2 -10070.33} C_VEL
LIN {X 0,Y 418.48,Z 236.358,A -85,B 0,C 180,E1 -10073.25,E2 -10073.25} C_VEL
LIN {X 0,Y 418.342,Z 236.374,A -85,B 0,C 180,E1 -10075.183,E2 -10075.183} C_VEL
LIN {X 0,Y 418.548,Z 236.351,A -85,B 0,C 180,E1 -10078.077,E2 -10078.077} C_VEL
LIN {X 0,Y 418.677,Z 236.335,A -85,B 0,C 180,E1 -10080.001,E2 -10080.001} C_VEL
LIN {X 0,Y 418.5,Z 236.353,A -85,B 0,C 180,E1 -10082.889,E2 -10082.889} C_VEL
LIN {X 0,Y 418.512,Z 236.356,A -85,B 0,C 180,E1 -10085.784,E2 -10085.784} C_VEL
LIN {X 0,Y 418.386,Z 236.368,A -85,B 0,C 180,E1 -10088.697,E2 -10088.697} C_VEL
LIN {X 0,Y 418.323,Z 236.379,A -85,B 0,C 180,E1 -10091.632,E2 -10091.632} C_VEL
LIN {X 0,Y 418.31,Z 236.378,A -85,B 0,C 180,E1 -10094.598,E2 -10094.598} C_VEL
LIN {X 0,Y 418.294,Z 236.383,A -85,B 0,C 180,E1 -10097.605,E2 -10097.605} C_VEL
LIN {X 0,Y 418.259,Z 236.385,A -85,B 0,C 180,E1 -10100.664,E2 -10100.664} C_VEL
LIN {X 0,Y 418.293,Z 236.382,A -85,B 0,C 180,E1 -10103.782,E2 -10103.782} C_VEL
LIN {X 0,Y 418.32,Z 236.379,A -85,B 0,C 180,E1 -10107.071,E2 -10107.071} C_VEL
LIN {X 0,Y 418.254,Z 236.384,A -85,B 0,C 180,E1 -10110.273,E2 -10110.273} C_VEL
LIN {X 0,Y 418.257,Z 236.386,A -85,B 0,C 180,E1 -10113.678,E2 -10113.678} C_VEL
LIN {X 0,Y 418.249,Z 236.389,A -85,B 0,C 180,E1 -10117.225,E2 -10117.225} C_VEL
LIN {X 0,Y 418.252,Z 236.388,A -85,B 0,C 180,E1 -10119.683,E2 -10119.683} C_VEL
LIN {X 0,Y 418.239,Z 236.39,A -85,B 0,C 180,E1 -10122.321,E2 -10122.321} C_VEL
LIN {X 0,Y 418.245,Z 236.386,A -85,B 0,C 180,E1 -10125.109,E2 -10125.109} C_VEL
LIN {X 0,Y 418.318,Z 236.53,A -85,B 0,C 180,E1 -10127.667,E2 -10127.667} C_VEL
LIN {X 0,Y 419.439,Z 243.002,A -85,B 0,C 180,E1 -10131.087,E2 -10131.087} C_VEL
LIN {X 0,Y 420.127,Z 247.662,A -85,B 0,C 180,E1 -10133.415,E2 -10133.415} C_VEL
LIN {X 0,Y 420.049,Z 251.708,A -85,B 0,C 180,E1 -10135.328,E2 -10135.328} C_VEL
LIN {X 0,Y 419.485,Z 257.97,A -85,B 0,C 180,E1 -10138.146,E2 -10138.146} C_VEL
LIN {X 0,Y 418.896,Z 265.476,A -85,B 0,C 180,E1 -10141.434,E2 -10141.434} C_VEL
LIN {X 0,Y 418.411,Z 273.037,A -85,B 0,C 180,E1 -10144.639,E2 -10144.639} C_VEL
LIN {X 0,Y 418.023,Z 280.253,A -85,B 0,C 180,E1 -10147.623,E2 -10147.623} C_VEL
LIN {X 0,Y 417.674,Z 288.302,A -85,B 0,C 180,E1 -10150.883,E2 -10150.883} C_VEL
LIN {X 0,Y 417.515,Z 293.152,A -85,B 0,C 180,E1 -10152.816,E2 -10152.816} C_VEL
LIN {X 0,Y 419.635,Z 307.263,A -85,B 0,C 180,E1 -10153.332,E2 -10153.332} C_VEL
LIN {X 0,Y 421.054,Z 319.738,A -85,B 0,C 180,E1 -10153.965,E2 -10153.965} C_VEL
LIN {X 0,Y 421.184,Z 324.97,A -85,B 0,C 180,E1 -10154.273,E2 -10154.273} C_VEL
LIN {X 0,Y 420.453,Z 337.111,A -85,B 0,C 180,E1 -10155.107,E2 -10155.107} C_VEL
LIN {X 0,Y 419.71,Z 348.099,A -85,B 0,C 180,E1 -10156.071,E2 -10156.071} C_VEL
LIN {X 0,Y 419.038,Z 358.03,A -85,B 0,C 180,E1 -10157.16,E2 -10157.16} C_VEL
LIN {X 0,Y 418.471,Z 367.061,A -85,B 0,C 180,E1 -10158.372,E2 -10158.372} C_VEL
LIN {X 0,Y 417.851,Z 375.891,A -85,B 0,C 180,E1 -10159.827,E2 -10159.827} C_VEL
LIN {X 0,Y 417.482,Z 382.95,A -85,B 0,C 180,E1 -10161.285,E2 -10161.285} C_VEL
LIN {X 0,Y 417.268,Z 388.597,A -85,B 0,C 180,E1 -10162.742,E2 -10162.742} C_VEL
LIN {X 0,Y 417.12,Z 393.03,A -85,B 0,C 180,E1 -10164.197,E2 -10164.197} C_VEL
LIN {X 0,Y 417.146,Z 395.373,A -85,B 0,C 180,E1 -10165.167,E2 -10165.167} C_VEL
LIN {X 0,Y 417.052,Z 397.272,A -85,B 0,C 180,E1 -10166.134,E2 -10166.134} C_VEL
LIN {X 0,Y 417.157,Z 398.724,A -85,B 0,C 180,E1 -10167.102,E2 -10167.102} C_VEL
LIN {X 0,Y 417.124,Z 399.737,A -85,B 0,C 180,E1 -10168.068,E2 -10168.068} C_VEL
LIN {X 0,Y 417.109,Z 400.356,A -85,B 0,C 180,E1 -10169.034,E2 -10169.034} C_VEL
LIN {X 0,Y 417.11,Z 400.583,A -85,B 0,C 180,E1 -10169.999,E2 -10169.999} C_VEL
LIN {X 0,Y 417.096,Z 400.38,A -85,B 0,C 180,E1 -10170.964,E2 -10170.964} C_VEL
LIN {X 0,Y 417.123,Z 399.764,A -85,B 0,C 180,E1 -10171.93,E2 -10171.93} C_VEL
LIN {X 0,Y 417.125,Z 398.752,A -85,B 0,C 180,E1 -10172.896,E2 -10172.896} C_VEL
LIN {X 0,Y 417.05,Z 397.333,A -85,B 0,C 180,E1 -10173.864,E2 -10173.864} C_VEL
LIN {X 0,Y 417.143,Z 394.362,A -85,B 0,C 180,E1 -10175.316,E2 -10175.316} C_VEL
LIN {X 0,Y 417.234,Z 390.345,A -85,B 0,C 180,E1 -10176.77,E2 -10176.77} C_VEL
LIN {X 0,Y 417.45,Z 384.189,A -85,B 0,C 180,E1 -10178.47,E2 -10178.47} C_VEL
LIN {X 0,Y 417.824,Z 377.461,A -85,B 0,C 180,E1 -10179.927,E2 -10179.927} C_VEL
LIN {X 0,Y 418.372,Z 369.143,A -85,B 0,C 180,E1 -10181.383,E2 -10181.383} C_VEL
LIN {X 0,Y 418.981,Z 360.661,A -85,B 0,C 180,E1 -10182.594,E2 -10182.594} C_VEL
LIN {X 0,Y 419.622,Z 350.465,A -85,B 0,C 180,E1 -10183.782,E2 -10183.782} C_VEL
LIN {X 0,Y 420.489,Z 338.529,A -85,B 0,C 180,E1 -10184.89,E2 -10184.89} C_VEL
LIN {X 0,Y 421.327,Z 326.978,A -85,B 0,C 180,E1 -10185.726,E2 -10185.726} C_VEL
LIN {X 0,Y 421.37,Z 320.903,A -85,B 0,C 180,E1 -10186.097,E2 -10186.097} C_VEL
LIN {X 0,Y 420.018,Z 307.527,A -85,B 0,C 180,E1 -10186.806,E2 -10186.806} C_VEL
LIN {X 0,Y 417.884,Z 294.378,A -85,B 0,C 180,E1 -10187.333,E2 -10187.333} C_VEL
LIN {X 0,Y 417.479,Z 292.048,A -85,B 0,C 180,E1 -10187.42,E2 -10187.42} C_VEL
LIN {X 0,Y 417.828,Z 283.87,A -85,B 0,C 180,E1 -10190.684,E2 -10190.684} C_VEL
LIN {X 0,Y 418.123,Z 276.302,A -85,B 0,C 180,E1 -10193.79,E2 -10193.79} C_VEL
LIN {X 0,Y 418.563,Z 268.814,A -85,B 0,C 180,E1 -10196.958,E2 -10196.958} C_VEL
LIN {X 0,Y 419.231,Z 260.256,A -85,B 0,C 180,E1 -10200.733,E2 -10200.733} C_VEL
LIN {X 0,Y 419.857,Z 254.245,A -85,B 0,C 180,E1 -10203.53,E2 -10203.53} C_VEL
LIN {X 0,Y 420.2,Z 249.533,A -85,B 0,C 180,E1 -10205.829,E2 -10205.829} C_VEL
LIN {X 0,Y 420.01,Z 246.2,A -85,B 0,C 180,E1 -10207.564,E2 -10207.564} C_VEL
LIN {X 0,Y 418.963,Z 240.176,A -85,B 0,C 180,E1 -10210.985,E2 -10210.985} C_VEL
LIN {X 0,Y 418.211,Z 236.395,A -85,B 0,C 180,E1 -10213.388,E2 -10213.388} C_VEL
LIN {X 0,Y 418.208,Z 236.394,A -85,B 0,C 180,E1 -10216.447,E2 -10216.447} C_VEL
LIN {X 0,Y 418.222,Z 236.392,A -85,B 0,C 180,E1 -10219.129,E2 -10219.129} C_VEL
LIN {X 0,Y 418.232,Z 236.391,A -85,B 0,C 180,E1 -10222.164,E2 -10222.164} C_VEL
LIN {X 0,Y 418.264,Z 236.387,A -85,B 0,C 180,E1 -10225.418,E2 -10225.418} C_VEL
LIN {X 0,Y 418.209,Z 236.393,A -85,B 0,C 180,E1 -10228.602,E2 -10228.602} C_VEL
LIN {X 0,Y 418.289,Z 236.383,A -85,B 0,C 180,E1 -10231.935,E2 -10231.935} C_VEL
LIN {X 0,Y 418.287,Z 236.383,A -85,B 0,C 180,E1 -10235.161,E2 -10235.161} C_VEL
LIN {X 0,Y 418.231,Z 236.39,A -85,B 0,C 180,E1 -10238.302,E2 -10238.302} C_VEL
LIN {X 0,Y 418.28,Z 236.384,A -85,B 0,C 180,E1 -10241.382,E2 -10241.382} C_VEL
LIN {X 0,Y 418.298,Z 236.38,A -85,B 0,C 180,E1 -10244.404,E2 -10244.404} C_VEL
LIN {X 0,Y 418.366,Z 236.374,A -85,B 0,C 180,E1 -10247.385,E2 -10247.385} C_VEL
LIN {X 0,Y 418.355,Z 236.375,A -85,B 0,C 180,E1 -10250.328,E2 -10250.328} C_VEL
LIN {X 0,Y 418.489,Z 236.358,A -85,B 0,C 180,E1 -10253.247,E2 -10253.247} C_VEL
LIN {X 0,Y 418.336,Z 236.378,A -85,B 0,C 180,E1 -10255.18,E2 -10255.18} C_VEL
LIN {X 0,Y 418.539,Z 236.352,A -85,B 0,C 180,E1 -10258.074,E2 -10258.074} C_VEL
LIN {X 0,Y 418.666,Z 236.336,A -85,B 0,C 180,E1 -10259.999,E2 -10259.999} C_VEL
LIN {X 0,Y 418.505,Z 236.357,A -85,B 0,C 180,E1 -10262.886,E2 -10262.886} C_VEL
LIN {X 0,Y 418.486,Z 236.357,A -85,B 0,C 180,E1 -10266.75,E2 -10266.75} C_VEL
LIN {X 0,Y 418.354,Z 236.376,A -85,B 0,C 180,E1 -10269.669,E2 -10269.669} C_VEL
LIN {X 0,Y 418.347,Z 236.377,A -85,B 0,C 180,E1 -10273.005,E2 -10273.005} C_VEL
LIN {X 0,Y 418.314,Z 236.385,A -85,B 0,C 180,E1 -10276.594,E2 -10276.594} C_VEL
LIN {X 0,Y 417.99,Z 236.423,A -85,B 0,C 180,E1 -10279.686,E2 -10279.686} C_VEL
LIN {X 0,Y 417.858,Z 239.035,A -85,B 0,C 180,E1 -10282.756,E2 -10282.756} C_VEL
LIN {X 0,Y 417.742,Z 242.061,A -85,B 0,C 180,E1 -10285.937,E2 -10285.937} C_VEL
LIN {X 0,Y 417.606,Z 245.182,A -85,B 0,C 180,E1 -10289.21,E2 -10289.21} C_VEL
LIN {X 0,Y 417.515,Z 248.567,A -85,B 0,C 180,E1 -10292.688,E2 -10292.688} C_VEL
LIN {X 0,Y 417.419,Z 251.563,A -85,B 0,C 180,E1 -10295.695,E2 -10295.695} C_VEL
LIN {X 0,Y 421.419,Z 266.762,A -85,B 0,C 180,E1 -10296.447,E2 -10296.447} C_VEL
LIN {X 0,Y 422.648,Z 273.272,A -85,B 0,C 180,E1 -10296.829,E2 -10296.829} C_VEL
LIN {X 0,Y 422.011,Z 285.007,A -85,B 0,C 180,E1 -10297.537,E2 -10297.537} C_VEL
LIN {X 0,Y 421.262,Z 296.395,A -85,B 0,C 180,E1 -10298.425,E2 -10298.425} C_VEL
LIN {X 0,Y 420.565,Z 307.477,A -85,B 0,C 180,E1 -10299.529,E2 -10299.529} C_VEL
LIN {X 0,Y 419.827,Z 317.336,A -85,B 0,C 180,E1 -10300.756,E2 -10300.756} C_VEL
LIN {X 0,Y 419.083,Z 326.269,A -85,B 0,C 180,E1 -10302.126,E2 -10302.126} C_VEL
LIN {X 0,Y 418.538,Z 333.497,A -85,B 0,C 180,E1 -10303.506,E2 -10303.506} C_VEL
LIN {X 0,Y 418.02,Z 340.071,A -85,B 0,C 180,E1 -10305.081,E2 -10305.081} C_VEL
LIN {X 0,Y 417.73,Z 344.412,A -85,B 0,C 180,E1 -10306.388,E2 -10306.388} C_VEL
LIN {X 0,Y 417.436,Z 348.085,A -85,B 0,C 180,E1 -10307.795,E2 -10307.795} C_VEL
LIN {X 0,Y 417.197,Z 350.932,A -85,B 0,C 180,E1 -10309.29,E2 -10309.29} C_VEL
LIN {X 0,Y 417.047,Z 352.803,A -85,B 0,C 180,E1 -10310.818,E2 -10310.818} C_VEL
LIN {X 0,Y 416.988,Z 353.71,A -85,B 0,C 180,E1 -10312.646,E2 -10312.646} C_VEL
LIN {X 0,Y 416.982,Z 353.486,A -85,B 0,C 180,E1 -10313.996,E2 -10313.996} C_VEL
LIN {X 0,Y 417.083,Z 352.141,A -85,B 0,C 180,E1 -10315.652,E2 -10315.652} C_VEL
LIN {X 0,Y 417.262,Z 349.461,A -85,B 0,C 180,E1 -10317.387,E2 -10317.387} C_VEL
LIN {X 0,Y 417.54,Z 345.346,A -85,B 0,C 180,E1 -10319.136,E2 -10319.136} C_VEL
LIN {X 0,Y 417.937,Z 339.275,A -85,B 0,C 180,E1 -10320.973,E2 -10320.973} C_VEL
LIN {X 0,Y 418.401,Z 332.969,A -85,B 0,C 180,E1 -10322.446,E2 -10322.446} C_VEL
LIN {X 0,Y 418.935,Z 325.327,A -85,B 0,C 180,E1 -10323.874,E2 -10323.874} C_VEL
LIN {X 0,Y 419.573,Z 316.212,A -85,B 0,C 180,E1 -10325.245,E2 -10325.245} C_VEL
LIN {X 0,Y 420.335,Z 306.036,A -85,B 0,C 180,E1 -10326.481,E2 -10326.481} C_VEL
LIN {X 0,Y 421.011,Z 294.948,A -85,B 0,C 180,E1 -10327.552,E2 -10327.552} C_VEL
LIN {X 0,Y 421.662,Z 282.625,A -85,B 0,C 180,E1 -10328.49,E2 -10328.49} C_VEL
LIN {X 0,Y 422.201,Z 271.815,A -85,B 0,C 180,E1 -10329.12,E2 -10329.12} C_VEL
LIN {X 0,Y 419.557,Z 259.408,A -85,B 0,C 180,E1 -10329.774,E2 -10329.774} C_VEL
LIN {X 0,Y 417.351,Z 250.429,A -85,B 0,C 180,E1 -10330.158,E2 -10330.158} C_VEL
LIN {X 0,Y 417.462,Z 246.759,A -85,B 0,C 180,E1 -10333.65,E2 -10333.65} C_VEL
LIN {X 0,Y 417.58,Z 242.814,A -85,B 0,C 180,E1 -10337.453,E2 -10337.453} C_VEL
LIN {X 0,Y 417.697,Z 238.927,A -85,B 0,C 180,E1 -10341.291,E2 -10341.291} C_VEL
LIN {X 0,Y 417.798,Z 236.962,A -85,B 0,C 180,E1 -10343.239,E2 -10343.239} C_VEL
LIN {X 0,Y 417.888,Z 236.432,A -85,B 0,C 180,E1 -10344.442,E2 -10344.442} C_VEL
LIN {X 0,Y 418.446,Z 236.361,A -85,B 0,C 180,E1 -10348.627,E2 -10348.627} C_VEL
LIN {X 0,Y 417.813,Z 236.444,A -85,B 0,C 180,E1 -10349.43,E2 -10349.43} C_VEL
LIN {X 0,Y 414.978,Z 236.794,A -85,B 0,C 180,E1 -10350.736,E2 -10350.736} C_VEL
LIN {X 0,Y 412.564,Z 237.095,A -85,B 0,C 180,E1 -10351.791,E2 -10351.791} C_VEL
LIN {X 0,Y 411.533,Z 237.222,A -85,B 0,C 180,E1 -10352.606,E2 -10352.606} C_VEL
LIN {X 0,Y 411.453,Z 237.233,A -85,B 0,C 180,E1 -10352.882,E2 -10352.882} C_VEL
LIN {X 0,Y 411.446,Z 237.235,A -85,B 0,C 180,E1 -10356.868,E2 -10356.868} C_VEL
LIN {X 0,Y 411.297,Z 237.252,A -85,B 0,C 180,E1 -10359.84,E2 -10359.84} C_VEL
LIN {X 0,Y 411.301,Z 237.255,A -85,B 0,C 180,E1 -10363.111,E2 -10363.111} C_VEL
LIN {X 0,Y 411.245,Z 237.262,A -85,B 0,C 180,E1 -10366.89,E2 -10366.89} C_VEL
LIN {X 0,Y 411.243,Z 237.258,A -85,B 0,C 180,E1 -10369.987,E2 -10369.987} C_VEL
LIN {X 0,Y 411.195,Z 237.268,A -85,B 0,C 180,E1 -10373.149,E2 -10373.149} C_VEL
LIN {X 0,Y 411.228,Z 237.262,A -85,B 0,C 180,E1 -10376.383,E2 -10376.383} C_VEL
LIN {X 0,Y 411.191,Z 237.264,A -85,B 0,C 180,E1 -10379.715,E2 -10379.715} C_VEL
LIN {X 0,Y 411.197,Z 237.266,A -85,B 0,C 180,E1 -10383.158,E2 -10383.158} C_VEL
LIN {X 0,Y 411.188,Z 237.268,A -85,B 0,C 180,E1 -10386.555,E2 -10386.555} C_VEL
LIN {X 0,Y 411.221,Z 237.261,A -85,B 0,C 180,E1 -10389.732,E2 -10389.732} C_VEL
LIN {X 0,Y 411.216,Z 237.262,A -85,B 0,C 180,E1 -10393.129,E2 -10393.129} C_VEL
LIN {X 0,Y 411.167,Z 237.268,A -85,B 0,C 180,E1 -10395.883,E2 -10395.883} C_VEL
LIN {X 0,Y 411.208,Z 237.262,A -85,B 0,C 180,E1 -10399.502,E2 -10399.502} C_VEL
LIN {X 0,Y 411.202,Z 237.265,A -85,B 0,C 180,E1 -10402.03,E2 -10402.03} C_VEL
LIN {X 0,Y 411.204,Z 237.263,A -85,B 0,C 180,E1 -10405.669,E2 -10405.669} C_VEL
LIN {X 0,Y 411.188,Z 237.265,A -85,B 0,C 180,E1 -10409.155,E2 -10409.155} C_VEL
LIN {X 0,Y 411.259,Z 237.258,A -85,B 0,C 180,E1 -10412.524,E2 -10412.524} C_VEL
LIN {X 0,Y 411.226,Z 237.261,A -85,B 0,C 180,E1 -10415.787,E2 -10415.787} C_VEL
LIN {X 0,Y 411.198,Z 237.264,A -85,B 0,C 180,E1 -10418.968,E2 -10418.968} C_VEL
LIN {X 0,Y 411.255,Z 237.26,A -85,B 0,C 180,E1 -10422.087,E2 -10422.087} C_VEL
LIN {X 0,Y 411.266,Z 237.255,A -85,B 0,C 180,E1 -10425.149,E2 -10425.149} C_VEL
LIN {X 0,Y 411.302,Z 237.254,A -85,B 0,C 180,E1 -10428.17,E2 -10428.17} C_VEL
LIN {X 0,Y 411.443,Z 237.235,A -85,B 0,C 180,E1 -10432.193,E2 -10432.193} C_VEL
LIN {X 0,Y 411.475,Z 237.232,A -85,B 0,C 180,E1 -10434.12,E2 -10434.12} C_VEL
LIN {X 0,Y 411.517,Z 237.226,A -85,B 0,C 180,E1 -10438.044,E2 -10438.044} C_VEL
LIN {X 0,Y 411.647,Z 237.21,A -85,B 0,C 180,E1 -10440.002,E2 -10440.002} C_VEL
LIN {X 0,Y 411.457,Z 237.231,A -85,B 0,C 180,E1 -10442.939,E2 -10442.939} C_VEL
LIN {X 0,Y 411.473,Z 237.232,A -85,B 0,C 180,E1 -10445.883,E2 -10445.883} C_VEL
LIN {X 0,Y 411.327,Z 237.247,A -85,B 0,C 180,E1 -10448.847,E2 -10448.847} C_VEL
LIN {X 0,Y 411.292,Z 237.255,A -85,B 0,C 180,E1 -10451.834,E2 -10451.834} C_VEL
LIN {X 0,Y 411.268,Z 237.256,A -85,B 0,C 180,E1 -10454.854,E2 -10454.854} C_VEL
LIN {X 0,Y 411.259,Z 237.258,A -85,B 0,C 180,E1 -10457.916,E2 -10457.916} C_VEL
LIN {X 0,Y 411.206,Z 237.265,A -85,B 0,C 180,E1 -10461.035,E2 -10461.035} C_VEL
LIN {X 0,Y 411.226,Z 237.259,A -85,B 0,C 180,E1 -10464.217,E2 -10464.217} C_VEL
LIN {X 0,Y 411.268,Z 237.258,A -85,B 0,C 180,E1 -10467.478,E2 -10467.478} C_VEL
LIN {X 0,Y 411.199,Z 237.265,A -85,B 0,C 180,E1 -10470.848,E2 -10470.848} C_VEL
LIN {X 0,Y 411.214,Z 237.262,A -85,B 0,C 180,E1 -10474.334,E2 -10474.334} C_VEL
LIN {X 0,Y 411.199,Z 237.263,A -85,B 0,C 180,E1 -10477.975,E2 -10477.975} C_VEL
LIN {X 0,Y 411.173,Z 237.27,A -85,B 0,C 180,E1 -10481.228,E2 -10481.228} C_VEL
LIN {X 0,Y 411.185,Z 237.267,A -85,B 0,C 180,E1 -10484.491,E2 -10484.491} C_VEL
LIN {X 0,Y 411.237,Z 237.258,A -85,B 0,C 180,E1 -10487.297,E2 -10487.297} C_VEL
LIN {X 0,Y 412.142,Z 242.461,A -85,B 0,C 180,E1 -10490.118,E2 -10490.118} C_VEL
LIN {X 0,Y 413.069,Z 248.225,A -85,B 0,C 180,E1 -10493.099,E2 -10493.099} C_VEL
LIN {X 0,Y 413.031,Z 252.778,A -85,B 0,C 180,E1 -10495.29,E2 -10495.29} C_VEL
LIN {X 0,Y 412.374,Z 259.652,A -85,B 0,C 180,E1 -10498.447,E2 -10498.447} C_VEL
LIN {X 0,Y 411.851,Z 266.431,A -85,B 0,C 180,E1 -10501.457,E2 -10501.457} C_VEL
LIN {X 0,Y 411.29,Z 274.419,A -85,B 0,C 180,E1 -10504.912,E2 -10504.912} C_VEL
LIN {X 0,Y 410.903,Z 281.525,A -85,B 0,C 180,E1 -10507.895,E2 -10507.895} C_VEL
LIN {X 0,Y 410.577,Z 289.066,A -85,B 0,C 180,E1 -10511.019,E2 -10511.019} C_VEL
LIN {X 0,Y 410.452,Z 292.947,A -85,B 0,C 180,E1 -10512.547,E2 -10512.547} C_VEL
LIN {X 0,Y 412.541,Z 306.338,A -85,B 0,C 180,E1 -10513.038,E2 -10513.038} C_VEL
LIN {X 0,Y 414.047,Z 319.77,A -85,B 0,C 180,E1 -10513.73,E2 -10513.73} C_VEL
LIN {X 0,Y 414.316,Z 324.595,A -85,B 0,C 180,E1 -10514.024,E2 -10514.024} C_VEL
LIN {X 0,Y 413.535,Z 336.492,A -85,B 0,C 180,E1 -10514.852,E2 -10514.852} C_VEL
LIN {X 0,Y 412.775,Z 347.534,A -85,B 0,C 180,E1 -10515.832,E2 -10515.832} C_VEL
LIN {X 0,Y 412.08,Z 357.735,A -85,B 0,C 180,E1 -10516.969,E2 -10516.969} C_VEL
LIN {X 0,Y 411.483,Z 366.563,A -85,B 0,C 180,E1 -10518.172,E2 -10518.172} C_VEL
LIN {X 0,Y 410.798,Z 375.409,A -85,B 0,C 180,E1 -10519.65,E2 -10519.65} C_VEL
LIN {X 0,Y 410.414,Z 382.491,A -85,B 0,C 180,E1 -10521.133,E2 -10521.133} C_VEL
LIN {X 0,Y 410.186,Z 388.151,A -85,B 0,C 180,E1 -10522.616,E2 -10522.616} C_VEL
LIN {X 0,Y 410.041,Z 392.597,A -85,B 0,C 180,E1 -10524.096,E2 -10524.096} C_VEL
LIN {X 0,Y 410.075,Z 394.946,A -85,B 0,C 180,E1 -10525.083,E2 -10525.083} C_VEL
LIN {X 0,Y 409.969,Z 396.85,A -85,B 0,C 180,E1 -10526.067,E2 -10526.067} C_VEL
LIN {X 0,Y 410.054,Z 398.31,A -85,B 0,C 180,E1 -10527.052,E2 -10527.052} C_VEL
LIN {X 0,Y 410.052,Z 399.329,A -85,B 0,C 180,E1 -10528.035,E2 -10528.035} C_VEL
LIN {X 0,Y 410.029,Z 399.951,A -85,B 0,C 180,E1 -10529.017,E2 -10529.017} C_VEL
LIN {X 0,Y 410.027,Z 400.181,A -85,B 0,C 180,E1 -10529.999,E2 -10529.999} C_VEL
LIN {X 0,Y 410.016,Z 399.986,A -85,B 0,C 180,E1 -10530.981,E2 -10530.981} C_VEL
LIN {X 0,Y 410.05,Z 399.373,A -85,B 0,C 180,E1 -10531.963,E2 -10531.963} C_VEL
LIN {X 0,Y 410.023,Z 398.361,A -85,B 0,C 180,E1 -10532.947,E2 -10532.947} C_VEL
LIN {X 0,Y 409.967,Z 396.947,A -85,B 0,C 180,E1 -10533.931,E2 -10533.931} C_VEL
LIN {X 0,Y 410.037,Z 393.982,A -85,B 0,C 180,E1 -10535.408,E2 -10535.408} C_VEL
LIN {X 0,Y 410.166,Z 389.977,A -85,B 0,C 180,E1 -10536.888,E2 -10536.888} C_VEL
LIN {X 0,Y 410.38,Z 383.84,A -85,B 0,C 180,E1 -10538.617,E2 -10538.617} C_VEL
LIN {X 0,Y 410.788,Z 377.134,A -85,B 0,C 180,E1 -10540.099,E2 -10540.099} C_VEL
